LIN {X 0,Y 573.014,Z 552.895,A -85,B 0,C 180,E1 -2253.868,E2 -2253.868} C_VEL
LIN {X 0,Y 572.963,Z 548.948,A -85,B 0,C 180,E1 -2254.926,E2 -2254.926} C_VEL
LIN {X 0,Y 573.068,Z 542.875,A -85,B 0,C 180,E1 -2256.16,E2 -2256.16} C_VEL
LIN {X 0,Y 573.12,Z 536.235,A -85,B 0,C 180,E1 -2257.221,E2 -2257.221} C_VEL
LIN {X 0,Y 573.192,Z 527.989,A -85,B 0,C 180,E1 -2258.284,E2 -2258.284} C_VEL
LIN {X 0,Y 573.32,Z 517.598,A -85,B 0,C 180,E1 -2259.348,E2 -2259.348} C_VEL
LIN {X 0,Y 573.431,Z 507.921,A -85,B 0,C 180,E1 -2260.148,E2 -2260.148} C_VEL
LIN {X 0,Y 573.55,Z 497.399,A -85,B 0,C 180,E1 -2260.855,E2 -2260.855} C_VEL
LIN {X 0,Y 573.653,Z 486.284,A -85,B 0,C 180,E1 -2261.447,E2 -2261.447} C_VEL
LIN {X 0,Y 573.72,Z 473.165,A -85,B 0,C 180,E1 -2261.975,E2 -2261.975} C_VEL
LIN {X 0,Y 573.814,Z 460.51,A -85,B 0,C 180,E1 -2262.332,E2 -2262.332} C_VEL
LIN {X 0,Y 573.909,Z 447.293,A -85,B 0,C 180,E1 -2262.554,E2 -2262.554} C_VEL
LIN {X 0,Y 573.91,Z 350.259,A -85,B 0,C 180,E1 -2263.776,E2 -2263.776} C_VEL
LIN {X 0,Y 573.399,Z 346.611,A -85,B 0,C 180,E1 -2263.851,E2 -2263.851} C_VEL
LIN {X 0,Y 573.569,Z 326.119,A -85,B 0,C 180,E1 -2266.727,E2 -2266.727} C_VEL
LIN {X 0,Y 573.804,Z 305.61,A -85,B 0,C 180,E1 -2269.646,E2 -2269.646} C_VEL
LIN {X 0,Y 574.03,Z 285.748,A -85,B 0,C 180,E1 -2272.495,E2 -2272.495} C_VEL
LIN {X 0,Y 573.588,Z 280.776,A -85,B 0,C 180,E1 -2273.226,E2 -2273.226} C_VEL
LIN {X 0,Y 573.253,Z 279.081,A -85,B 0,C 180,E1 -2273.497,E2 -2273.497} C_VEL
LIN {X 0,Y 573.261,Z 279.08,A -85,B 0,C 180,E1 -2276.19,E2 -2276.19} C_VEL
LIN {X 0,Y 573.237,Z 279.078,A -85,B 0,C 180,E1 -2278.564,E2 -2278.564} C_VEL
LIN {X 0,Y 573.227,Z 279.076,A -85,B 0,C 180,E1 -2280.993,E2 -2280.993} C_VEL
LIN {X 0,Y 573.265,Z 279.071,A -85,B 0,C 180,E1 -2283.524,E2 -2283.524} C_VEL
LIN {X 0,Y 573.216,Z 279.083,A -85,B 0,C 180,E1 -2286.051,E2 -2286.051} C_VEL
LIN {X 0,Y 573.241,Z 279.079,A -85,B 0,C 180,E1 -2288.701,E2 -2288.701} C_VEL
LIN {X 0,Y 573.23,Z 279.075,A -85,B 0,C 180,E1 -2291.593,E2 -2291.593} C_VEL
LIN {X 0,Y 573.222,Z 279.082,A -85,B 0,C 180,E1 -2294.334,E2 -2294.334} C_VEL
LIN {X 0,Y 573.241,Z 279.074,A -85,B 0,C 180,E1 -2297.358,E2 -2297.358} C_VEL
LIN {X 0,Y 573.239,Z 279.077,A -85,B 0,C 180,E1 -2300.392,E2 -2300.392} C_VEL
LIN {X 0,Y 573.252,Z 279.078,A -85,B 0,C 180,E1 -2303.077,E2 -2303.077} C_VEL
LIN {X 0,Y 573.266,Z 279.07,A -85,B 0,C 180,E1 -2305.671,E2 -2305.671} C_VEL
LIN {X 0,Y 573.239,Z 279.074,A -85,B 0,C 180,E1 -2308.184,E2 -2308.184} C_VEL
LIN {X 0,Y 573.263,Z 279.073,A -85,B 0,C 180,E1 -2310.634,E2 -2310.634} C_VEL
LIN {X 0,Y 573.249,Z 279.08,A -85,B 0,C 180,E1 -2313.024,E2 -2313.024} C_VEL
LIN {X 0,Y 573.273,Z 279.077,A -85,B 0,C 180,E1 -2315.366,E2 -2315.366} C_VEL
LIN {X 0,Y 573.227,Z 279.075,A -85,B 0,C 180,E1 -2318.419,E2 -2318.419} C_VEL
LIN {X 0,Y 573.277,Z 279.069,A -85,B 0,C 180,E1 -2320.728,E2 -2320.728} C_VEL
LIN {X 0,Y 573.249,Z 279.08,A -85,B 0,C 180,E1 -2323.622,E2 -2323.622} C_VEL
LIN {X 0,Y 573.271,Z 279.075,A -85,B 0,C 180,E1 -2325.807,E2 -2325.807} C_VEL
LIN {X 0,Y 573.26,Z 279.07,A -85,B 0,C 180,E1 -2328.745,E2 -2328.745} C_VEL
LIN {X 0,Y 573.281,Z 279.074,A -85,B 0,C 180,E1 -2331.54,E2 -2331.54} C_VEL
LIN {X 0,Y 573.288,Z 279.068,A -85,B 0,C 180,E1 -2334.372,E2 -2334.372} C_VEL
LIN {X 0,Y 573.309,Z 279.074,A -85,B 0,C 180,E1 -2337.892,E2 -2337.892} C_VEL
LIN {X 0,Y 573.327,Z 279.063,A -85,B 0,C 180,E1 -2340.702,E2 -2340.702} C_VEL
LIN {X 0,Y 573.236,Z 279.074,A -85,B 0,C 180,E1 -2343.514,E2 -2343.514} C_VEL
LIN {X 0,Y 573.288,Z 279.069,A -85,B 0,C 180,E1 -2345.628,E2 -2345.628} C_VEL
LIN {X 0,Y 573.281,Z 279.075,A -85,B 0,C 180,E1 -2348.459,E2 -2348.459} C_VEL
LIN {X 0,Y 573.269,Z 279.069,A -85,B 0,C 180,E1 -2351.312,E2 -2351.312} C_VEL
LIN {X 0,Y 573.279,Z 279.079,A -85,B 0,C 180,E1 -2354.424,E2 -2354.424} C_VEL
LIN {X 0,Y 573.256,Z 279.073,A -85,B 0,C 180,E1 -2357.112,E2 -2357.112} C_VEL
LIN {X 0,Y 573.25,Z 279.074,A -85,B 0,C 180,E1 -2360.077,E2 -2360.077} C_VEL
LIN {X 0,Y 573.232,Z 279.078,A -85,B 0,C 180,E1 -2363.099,E2 -2363.099} C_VEL
LIN {X 0,Y 573.248,Z 279.076,A -85,B 0,C 180,E1 -2364.382,E2 -2364.382} C_VEL
LIN {X 0,Y 572.62,Z 279.161,A -85,B 0,C 180,E1 -2364.969,E2 -2364.969} C_VEL
LIN {X 0,Y 569.779,Z 279.516,A -85,B 0,C 180,E1 -2365.92,E2 -2365.92} C_VEL
LIN {X 0,Y 567.347,Z 279.815,A -85,B 0,C 180,E1 -2366.686,E2 -2366.686} C_VEL
LIN {X 0,Y 566.292,Z 279.942,A -85,B 0,C 180,E1 -2367.277,E2 -2367.277} C_VEL
LIN {X 0,Y 566.201,Z 279.951,A -85,B 0,C 180,E1 -2367.477,E2 -2367.477} C_VEL
LIN {X 0,Y 566.199,Z 279.95,A -85,B 0,C 180,E1 -2369.769,E2 -2369.769} C_VEL
LIN {X 0,Y 566.201,Z 279.951,A -85,B 0,C 180,E1 -2372.43,E2 -2372.43} C_VEL
LIN {X 0,Y 566.179,Z 279.961,A -85,B 0,C 180,E1 -2374.99,E2 -2374.99} C_VEL
LIN {X 0,Y 566.195,Z 279.957,A -85,B 0,C 180,E1 -2377.461,E2 -2377.461} C_VEL
LIN {X 0,Y 566.206,Z 279.949,A -85,B 0,C 180,E1 -2380.199,E2 -2380.199} C_VEL
LIN {X 0,Y 566.2,Z 279.956,A -85,B 0,C 180,E1 -2383.054,E2 -2383.054} C_VEL
LIN {X 0,Y 566.193,Z 279.953,A -85,B 0,C 180,E1 -2386.049,E2 -2386.049} C_VEL
LIN {X 0,Y 566.203,Z 279.955,A -85,B 0,C 180,E1 -2389.215,E2 -2389.215} C_VEL
LIN {X 0,Y 566.185,Z 279.962,A -85,B 0,C 180,E1 -2391.637,E2 -2391.637} C_VEL
LIN {X 0,Y 566.162,Z 279.957,A -85,B 0,C 180,E1 -2394.308,E2 -2394.308} C_VEL
LIN {X 0,Y 566.205,Z 279.951,A -85,B 0,C 180,E1 -2396.897,E2 -2396.897} C_VEL
LIN {X 0,Y 566.181,Z 279.958,A -85,B 0,C 180,E1 -2399.407,E2 -2399.407} C_VEL
LIN {X 0,Y 566.242,Z 280.056,A -85,B 0,C 180,E1 -2400.897,E2 -2400.897} C_VEL
LIN {X 0,Y 566.45,Z 286.564,A -85,B 0,C 180,E1 -2402.072,E2 -2402.072} C_VEL
LIN {X 0,Y 566.262,Z 302.821,A -85,B 0,C 180,E1 -2405.04,E2 -2405.04} C_VEL
LIN {X 0,Y 566.202,Z 308.373,A -85,B 0,C 180,E1 -2406.045,E2 -2406.045} C_VEL
LIN {X 0,Y 567.204,Z 314.789,A -85,B 0,C 180,E1 -2406.161,E2 -2406.161} C_VEL
LIN {X 0,Y 566.892,Z 414.942,A -85,B 0,C 180,E1 -2407.447,E2 -2407.447} C_VEL
LIN {X 0,Y 566.74,Z 428.708,A -85,B 0,C 180,E1 -2407.776,E2 -2407.776} C_VEL
LIN {X 0,Y 566.676,Z 440.788,A -85,B 0,C 180,E1 -2408.209,E2 -2408.209} C_VEL
LIN {X 0,Y 566.58,Z 452.966,A -85,B 0,C 180,E1 -2408.798,E2 -2408.798} C_VEL
LIN {X 0,Y 566.416,Z 463.929,A -85,B 0,C 180,E1 -2409.481,E2 -2409.481} C_VEL
LIN {X 0,Y 566.302,Z 474.815,A -85,B 0,C 180,E1 -2410.328,E2 -2410.328} C_VEL
LIN {X 0,Y 566.23,Z 483.591,A -85,B 0,C 180,E1 -2411.173,E2 -2411.173} C_VEL
LIN {X 0,Y 566.102,Z 491.649,A -85,B 0,C 180,E1 -2412.105,E2 -2412.105} C_VEL
LIN {X 0,Y 566.039,Z 499.147,A -85,B 0,C 180,E1 -2413.176,E2 -2413.176} C_VEL
LIN {X 0,Y 565.951,Z 504.676,A -85,B 0,C 180,E1 -2414.145,E2 -2414.145} C_VEL
LIN {X 0,Y 565.943,Z 509.72,A -85,B 0,C 180,E1 -2415.252,E2 -2415.252} C_VEL
LIN {X 0,Y 565.898,Z 513.562,A -85,B 0,C 180,E1 -2416.351,E2 -2416.351} C_VEL
LIN {X 0,Y 565.86,Z 515.527,A -85,B 0,C 180,E1 -2417.082,E2 -2417.082} C_VEL
LIN {X 0,Y 565.869,Z 517.042,A -85,B 0,C 180,E1 -2417.811,E2 -2417.811} C_VEL
LIN {X 0,Y 565.901,Z 518.433,A -85,B 0,C 180,E1 -2418.846,E2 -2418.846} C_VEL
LIN {X 0,Y 565.882,Z 518.993,A -85,B 0,C 180,E1 -2419.987,E2 -2419.987} C_VEL
LIN {X 0,Y 565.829,Z 518.818,A -85,B 0,C 180,E1 -2420.708,E2 -2420.708} C_VEL
LIN {X 0,Y 565.851,Z 518.23,A -85,B 0,C 180,E1 -2421.428,E2 -2421.428} C_VEL
LIN {X 0,Y 565.876,Z 517.248,A -85,B 0,C 180,E1 -2422.148,E2 -2422.148} C_VEL
LIN {X 0,Y 565.946,Z 514.44,A -85,B 0,C 180,E1 -2423.44,E2 -2423.44} C_VEL
LIN {X 0,Y 565.921,Z 510.451,A -85,B 0,C 180,E1 -2424.655,E2 -2424.655} C_VEL
LIN {X 0,Y 565.964,Z 505.778,A -85,B 0,C 180,E1 -2425.727,E2 -2425.727} C_VEL
LIN {X 0,Y 566.002,Z 498.771,A -85,B 0,C 180,E1 -2426.975,E2 -2426.975} C_VEL
LIN {X 0,Y 566.065,Z 491.207,A -85,B 0,C 180,E1 -2428.043,E2 -2428.043} C_VEL
LIN {X 0,Y 566.211,Z 481.731,A -85,B 0,C 180,E1 -2429.111,E2 -2429.111} C_VEL
LIN {X 0,Y 566.297,Z 472.006,A -85,B 0,C 180,E1 -2430,E2 -2430} C_VEL
LIN {X 0,Y 566.443,Z 461.142,A -85,B 0,C 180,E1 -2430.799,E2 -2430.799} C_VEL
LIN {X 0,Y 566.641,Z 448.809,A -85,B 0,C 180,E1 -2431.51,E2 -2431.51} C_VEL
LIN {X 0,Y 566.743,Z 436.745,A -85,B 0,C 180,E1 -2432.043,E2 -2432.043} C_VEL
LIN {X 0,Y 566.815,Z 424.109,A -85,B 0,C 180,E1 -2432.442,E2 -2432.442} C_VEL
LIN {X 0,Y 566.945,Z 410.737,A -85,B 0,C 180,E1 -2432.708,E2 -2432.708} C_VEL
LIN {X 0,Y 567.094,Z 313.951,A -85,B 0,C 180,E1 -2433.943,E2 -2433.943} C_VEL
LIN {X 0,Y 566.199,Z 308.359,A -85,B 0,C 180,E1 -2434.048,E2 -2434.048} C_VEL
LIN {X 0,Y 566.374,Z 295.33,A -85,B 0,C 180,E1 -2436.412,E2 -2436.412} C_VEL
LIN {X 0,Y 566.401,Z 281.613,A -85,B 0,C 180,E1 -2438.922,E2 -2438.922} C_VEL
LIN {X 0,Y 566.187,Z 279.958,A -85,B 0,C 180,E1 -2439.241,E2 -2439.241} C_VEL
LIN {X 0,Y 566.192,Z 279.953,A -85,B 0,C 180,E1 -2441.455,E2 -2441.455} C_VEL
LIN {X 0,Y 566.213,Z 279.956,A -85,B 0,C 180,E1 -2444.497,E2 -2444.497} C_VEL
LIN {X 0,Y 566.17,Z 279.954,A -85,B 0,C 180,E1 -2447.332,E2 -2447.332} C_VEL
LIN {X 0,Y 566.2,Z 279.959,A -85,B 0,C 180,E1 -2450.337,E2 -2450.337} C_VEL
LIN {X 0,Y 566.163,Z 279.955,A -85,B 0,C 180,E1 -2453.279,E2 -2453.279} C_VEL
LIN {X 0,Y 566.169,Z 279.954,A -85,B 0,C 180,E1 -2455.75,E2 -2455.75} C_VEL
LIN {X 0,Y 566.149,Z 279.96,A -85,B 0,C 180,E1 -2458.192,E2 -2458.192} C_VEL
LIN {X 0,Y 566.177,Z 279.958,A -85,B 0,C 180,E1 -2461.074,E2 -2461.074} C_VEL
LIN {X 0,Y 566.192,Z 279.951,A -85,B 0,C 180,E1 -2463.731,E2 -2463.731} C_VEL
LIN {X 0,Y 566.193,Z 279.956,A -85,B 0,C 180,E1 -2466.569,E2 -2466.569} C_VEL
LIN {X 0,Y 566.204,Z 279.95,A -85,B 0,C 180,E1 -2469.684,E2 -2469.684} C_VEL
LIN {X 0,Y 566.166,Z 279.954,A -85,B 0,C 180,E1 -2472.09,E2 -2472.09} C_VEL
LIN {X 0,Y 566.161,Z 279.964,A -85,B 0,C 180,E1 -2475.036,E2 -2475.036} C_VEL
LIN {X 0,Y 566.18,Z 279.953,A -85,B 0,C 180,E1 -2477.91,E2 -2477.91} C_VEL
LIN {X 0,Y 566.203,Z 279.952,A -85,B 0,C 180,E1 -2480.725,E2 -2480.725} C_VEL
LIN {X 0,Y 566.175,Z 279.957,A -85,B 0,C 180,E1 -2483.788,E2 -2483.788} C_VEL
LIN {X 0,Y 566.203,Z 279.95,A -85,B 0,C 180,E1 -2486.265,E2 -2486.265} C_VEL
LIN {X 0,Y 566.18,Z 279.955,A -85,B 0,C 180,E1 -2488.923,E2 -2488.923} C_VEL
LIN {X 0,Y 566.178,Z 279.958,A -85,B 0,C 180,E1 -2491.856,E2 -2491.856} C_VEL
LIN {X 0,Y 566.203,Z 279.951,A -85,B 0,C 180,E1 -2494.251,E2 -2494.251} C_VEL
LIN {X 0,Y 566.16,Z 279.955,A -85,B 0,C 180,E1 -2496.719,E2 -2496.719} C_VEL
LIN {X 0,Y 566.198,Z 279.959,A -85,B 0,C 180,E1 -2499.662,E2 -2499.662} C_VEL
LIN {X 0,Y 566.192,Z 279.951,A -85,B 0,C 180,E1 -2502.668,E2 -2502.668} C_VEL
LIN {X 0,Y 566.211,Z 279.954,A -85,B 0,C 180,E1 -2505.626,E2 -2505.626} C_VEL
LIN {X 0,Y 566.225,Z 279.948,A -85,B 0,C 180,E1 -2508.675,E2 -2508.675} C_VEL
LIN {X 0,Y 566.218,Z 279.949,A -85,B 0,C 180,E1 -2511.434,E2 -2511.434} C_VEL
LIN {X 0,Y 566.253,Z 279.952,A -85,B 0,C 180,E1 -2514.302,E2 -2514.302} C_VEL
LIN {X 0,Y 566.268,Z 279.946,A -85,B 0,C 180,E1 -2517.866,E2 -2517.866} C_VEL
LIN {X 0,Y 566.299,Z 279.942,A -85,B 0,C 180,E1 -2520.711,E2 -2520.711} C_VEL
LIN {X 0,Y 566.269,Z 279.945,A -85,B 0,C 180,E1 -2522.846,E2 -2522.846} C_VEL
LIN {X 0,Y 566.249,Z 279.944,A -85,B 0,C 180,E1 -2525.699,E2 -2525.699} C_VEL
LIN {X 0,Y 566.239,Z 279.956,A -85,B 0,C 180,E1 -2528.566,E2 -2528.566} C_VEL
LIN {X 0,Y 566.243,Z 279.945,A -85,B 0,C 180,E1 -2531.454,E2 -2531.454} C_VEL
LIN {X 0,Y 566.225,Z 279.954,A -85,B 0,C 180,E1 -2534.507,E2 -2534.507} C_VEL
LIN {X 0,Y 566.191,Z 279.953,A -85,B 0,C 180,E1 -2537.332,E2 -2537.332} C_VEL
LIN {X 0,Y 566.205,Z 279.952,A -85,B 0,C 180,E1 -2540.338,E2 -2540.338} C_VEL
LIN {X 0,Y 566.182,Z 279.955,A -85,B 0,C 180,E1 -2543.404,E2 -2543.404} C_VEL
LIN {X 0,Y 566.218,Z 279.948,A -85,B 0,C 180,E1 -2545.749,E2 -2545.749} C_VEL
LIN {X 0,Y 566.195,Z 279.951,A -85,B 0,C 180,E1 -2548.203,E2 -2548.203} C_VEL
LIN {X 0,Y 566.187,Z 279.954,A -85,B 0,C 180,E1 -2550.593,E2 -2550.593} C_VEL
LIN {X 0,Y 566.223,Z 279.956,A -85,B 0,C 180,E1 -2553.102,E2 -2553.102} C_VEL
LIN {X 0,Y 566.2,Z 279.95,A -85,B 0,C 180,E1 -2556.216,E2 -2556.216} C_VEL
LIN {X 0,Y 566.216,Z 279.957,A -85,B 0,C 180,E1 -2559.274,E2 -2559.274} C_VEL
LIN {X 0,Y 566.209,Z 279.95,A -85,B 0,C 180,E1 -2562.088,E2 -2562.088} C_VEL
LIN {X 0,Y 566.169,Z 279.957,A -85,B 0,C 180,E1 -2565.037,E2 -2565.037} C_VEL
LIN {X 0,Y 566.215,Z 279.951,A -85,B 0,C 180,E1 -2568.137,E2 -2568.137} C_VEL
LIN {X 0,Y 566.211,Z 279.949,A -85,B 0,C 180,E1 -2570.727,E2 -2570.727} C_VEL
LIN {X 0,Y 566.182,Z 279.963,A -85,B 0,C 180,E1 -2573.789,E2 -2573.789} C_VEL
LIN {X 0,Y 566.21,Z 279.952,A -85,B 0,C 180,E1 -2576.267,E2 -2576.267} C_VEL
LIN {X 0,Y 566.189,Z 279.951,A -85,B 0,C 180,E1 -2578.924,E2 -2578.924} C_VEL
LIN {X 0,Y 566.229,Z 279.957,A -85,B 0,C 180,E1 -2581.859,E2 -2581.859} C_VEL
LIN {X 0,Y 566.237,Z 279.948,A -85,B 0,C 180,E1 -2585.04,E2 -2585.04} C_VEL
LIN {X 0,Y 566.24,Z 280.067,A -85,B 0,C 180,E1 -2586.381,E2 -2586.381} C_VEL
LIN {X 0,Y 567.09,Z 285.538,A -85,B 0,C 180,E1 -2587.215,E2 -2587.215} C_VEL
LIN {X 0,Y 566.868,Z 306.731,A -85,B 0,C 180,E1 -2590.274,E2 -2590.274} C_VEL
LIN {X 0,Y 566.599,Z 327.553,A -85,B 0,C 180,E1 -2593.267,E2 -2593.267} C_VEL
LIN {X 0,Y 566.389,Z 346.617,A -85,B 0,C 180,E1 -2595.975,E2 -2595.975} C_VEL
LIN {X 0,Y 567.201,Z 352.33,A -85,B 0,C 180,E1 -2596.084,E2 -2596.084} C_VEL
LIN {X 0,Y 566.953,Z 454.975,A -85,B 0,C 180,E1 -2597.403,E2 -2597.403} C_VEL
LIN {X 0,Y 566.837,Z 468.237,A -85,B 0,C 180,E1 -2597.719,E2 -2597.719} C_VEL
LIN {X 0,Y 566.722,Z 480.39,A -85,B 0,C 180,E1 -2598.148,E2 -2598.148} C_VEL
LIN {X 0,Y 566.626,Z 492.163,A -85,B 0,C 180,E1 -2598.709,E2 -2598.709} C_VEL
LIN {X 0,Y 566.458,Z 504.206,A -85,B 0,C 180,E1 -2599.456,E2 -2599.456} C_VEL
LIN {X 0,Y 566.32,Z 514.609,A -85,B 0,C 180,E1 -2600.266,E2 -2600.266} C_VEL
LIN {X 0,Y 566.205,Z 523.088,A -85,B 0,C 180,E1 -2601.075,E2 -2601.075} C_VEL
LIN {X 0,Y 566.111,Z 530.965,A -85,B 0,C 180,E1 -2601.972,E2 -2601.972} C_VEL
LIN {X 0,Y 566.003,Z 538.625,A -85,B 0,C 180,E1 -2603.047,E2 -2603.047} C_VEL
LIN {X 0,Y 566.004,Z 545.682,A -85,B 0,C 180,E1 -2604.3,E2 -2604.3} C_VEL
LIN {X 0,Y 565.933,Z 550.374,A -85,B 0,C 180,E1 -2605.371,E2 -2605.371} C_VEL
LIN {X 0,Y 565.926,Z 553.959,A -85,B 0,C 180,E1 -2606.44,E2 -2606.44} C_VEL
LIN {X 0,Y 565.878,Z 555.809,A -85,B 0,C 180,E1 -2607.153,E2 -2607.153} C_VEL
LIN {X 0,Y 565.845,Z 558.185,A -85,B 0,C 180,E1 -2608.577,E2 -2608.577} C_VEL
LIN {X 0,Y 565.839,Z 559,A -85,B 0,C 180,E1 -2610,E2 -2610} C_VEL
LIN {X 0,Y 565.845,Z 558.185,A -85,B 0,C 180,E1 -2611.424,E2 -2611.424} C_VEL
LIN {X 0,Y 565.878,Z 555.809,A -85,B 0,C 180,E1 -2612.848,E2 -2612.848} C_VEL
LIN {X 0,Y 565.926,Z 552.895,A -85,B 0,C 180,E1 -2613.917,E2 -2613.917} C_VEL
LIN {X 0,Y 565.878,Z 548.947,A -85,B 0,C 180,E1 -2614.988,E2 -2614.988} C_VEL
LIN {X 0,Y 565.994,Z 542.875,A -85,B 0,C 180,E1 -2616.238,E2 -2616.238} C_VEL
LIN {X 0,Y 566.052,Z 536.235,A -85,B 0,C 180,E1 -2617.312,E2 -2617.312} C_VEL
LIN {X 0,Y 566.141,Z 527.989,A -85,B 0,C 180,E1 -2618.388,E2 -2618.388} C_VEL
LIN {X 0,Y 566.254,Z 519.536,A -85,B 0,C 180,E1 -2619.285,E2 -2619.285} C_VEL
LIN {X 0,Y 566.416,Z 509.093,A -85,B 0,C 180,E1 -2620.184,E2 -2620.184} C_VEL
LIN {X 0,Y 566.571,Z 497.699,A -85,B 0,C 180,E1 -2620.971,E2 -2620.971} C_VEL
LIN {X 0,Y 566.693,Z 485.881,A -85,B 0,C 180,E1 -2621.608,E2 -2621.608} C_VEL
LIN {X 0,Y 566.79,Z 473.163,A -85,B 0,C 180,E1 -2622.124,E2 -2622.124} C_VEL
LIN {X 0,Y 566.877,Z 460.509,A -85,B 0,C 180,E1 -2622.485,E2 -2622.485} C_VEL
LIN {X 0,Y 566.977,Z 447.293,A -85,B 0,C 180,E1 -2622.71,E2 -2622.71} C_VEL
LIN {X 0,Y 567.066,Z 351.263,A -85,B 0,C 180,E1 -2623.933,E2 -2623.933} C_VEL
LIN {X 0,Y 566.407,Z 346.611,A -85,B 0,C 180,E1 -2624.025,E2 -2624.025} C_VEL
LIN {X 0,Y 566.607,Z 324.039,A -85,B 0,C 180,E1 -2627.238,E2 -2627.238} C_VEL
LIN {X 0,Y 566.869,Z 303.946,A -85,B 0,C 180,E1 -2630.123,E2 -2630.123} C_VEL
LIN {X 0,Y 567.055,Z 285.451,A -85,B 0,C 180,E1 -2632.787,E2 -2632.787} C_VEL
LIN {X 0,Y 566.215,Z 279.958,A -85,B 0,C 180,E1 -2633.645,E2 -2633.645} C_VEL
LIN {X 0,Y 566.21,Z 279.958,A -85,B 0,C 180,E1 -2635.749,E2 -2635.749} C_VEL
LIN {X 0,Y 566.206,Z 279.96,A -85,B 0,C 180,E1 -2638.202,E2 -2638.202} C_VEL
LIN {X 0,Y 566.193,Z 279.953,A -85,B 0,C 180,E1 -2641.076,E2 -2641.076} C_VEL
LIN {X 0,Y 566.213,Z 279.951,A -85,B 0,C 180,E1 -2643.734,E2 -2643.734} C_VEL
LIN {X 0,Y 566.201,Z 279.957,A -85,B 0,C 180,E1 -2646.57,E2 -2646.57} C_VEL
LIN {X 0,Y 566.215,Z 279.949,A -85,B 0,C 180,E1 -2649.685,E2 -2649.685} C_VEL
LIN {X 0,Y 566.202,Z 279.955,A -85,B 0,C 180,E1 -2652.917,E2 -2652.917} C_VEL
LIN {X 0,Y 566.194,Z 279.953,A -85,B 0,C 180,E1 -2656.049,E2 -2656.049} C_VEL
LIN {X 0,Y 566.204,Z 279.952,A -85,B 0,C 180,E1 -2659.214,E2 -2659.214} C_VEL
LIN {X 0,Y 566.186,Z 279.952,A -85,B 0,C 180,E1 -2661.637,E2 -2661.637} C_VEL
LIN {X 0,Y 566.162,Z 279.957,A -85,B 0,C 180,E1 -2664.308,E2 -2664.308} C_VEL
LIN {X 0,Y 566.219,Z 279.957,A -85,B 0,C 180,E1 -2666.898,E2 -2666.898} C_VEL
LIN {X 0,Y 566.18,Z 279.957,A -85,B 0,C 180,E1 -2669.407,E2 -2669.407} C_VEL
LIN {X 0,Y 566.21,Z 279.95,A -85,B 0,C 180,E1 -2671.857,E2 -2671.857} C_VEL
LIN {X 0,Y 566.212,Z 279.948,A -85,B 0,C 180,E1 -2674.251,E2 -2674.251} C_VEL
LIN {X 0,Y 566.172,Z 279.956,A -85,B 0,C 180,E1 -2676.718,E2 -2676.718} C_VEL
LIN {X 0,Y 566.212,Z 279.954,A -85,B 0,C 180,E1 -2679.663,E2 -2679.663} C_VEL
LIN {X 0,Y 566.198,Z 279.95,A -85,B 0,C 180,E1 -2682.668,E2 -2682.668} C_VEL
LIN {X 0,Y 566.232,Z 279.955,A -85,B 0,C 180,E1 -2685.627,E2 -2685.627} C_VEL
LIN {X 0,Y 566.232,Z 279.945,A -85,B 0,C 180,E1 -2688.675,E2 -2688.675} C_VEL
LIN {X 0,Y 566.225,Z 279.951,A -85,B 0,C 180,E1 -2691.434,E2 -2691.434} C_VEL
LIN {X 0,Y 566.256,Z 279.945,A -85,B 0,C 180,E1 -2694.302,E2 -2694.302} C_VEL
LIN {X 0,Y 566.28,Z 279.949,A -85,B 0,C 180,E1 -2697.866,E2 -2697.866} C_VEL
LIN {X 0,Y 566.298,Z 279.938,A -85,B 0,C 180,E1 -2700.711,E2 -2700.711} C_VEL
LIN {X 0,Y 566.269,Z 279.941,A -85,B 0,C 180,E1 -2702.845,E2 -2702.845} C_VEL
LIN {X 0,Y 566.256,Z 279.945,A -85,B 0,C 180,E1 -2705.698,E2 -2705.698} C_VEL
LIN {X 0,Y 566.225,Z 279.952,A -85,B 0,C 180,E1 -2708.566,E2 -2708.566} C_VEL
LIN {X 0,Y 566.24,Z 279.945,A -85,B 0,C 180,E1 -2711.454,E2 -2711.454} C_VEL
LIN {X 0,Y 566.232,Z 279.956,A -85,B 0,C 180,E1 -2714.507,E2 -2714.507} C_VEL
LIN {X 0,Y 566.197,Z 279.951,A -85,B 0,C 180,E1 -2717.332,E2 -2717.332} C_VEL
LIN {X 0,Y 566.211,Z 279.954,A -85,B 0,C 180,E1 -2720.337,E2 -2720.337} C_VEL
LIN {X 0,Y 566.187,Z 279.953,A -85,B 0,C 180,E1 -2723.404,E2 -2723.404} C_VEL
LIN {X 0,Y 566.212,Z 279.948,A -85,B 0,C 180,E1 -2725.749,E2 -2725.749} C_VEL
LIN {X 0,Y 566.201,Z 279.951,A -85,B 0,C 180,E1 -2727.477,E2 -2727.477} C_VEL
LIN {X 0,Y 565.521,Z 280.036,A -85,B 0,C 180,E1 -2728.071,E2 -2728.071} C_VEL
LIN {X 0,Y 562.655,Z 280.4,A -85,B 0,C 180,E1 -2729.034,E2 -2729.034} C_VEL
LIN {X 0,Y 560.246,Z 280.696,A -85,B 0,C 180,E1 -2729.81,E2 -2729.81} C_VEL
LIN {X 0,Y 559.218,Z 280.822,A -85,B 0,C 180,E1 -2730.409,E2 -2730.409} C_VEL
LIN {X 0,Y 559.138,Z 280.833,A -85,B 0,C 180,E1 -2730.611,E2 -2730.611} C_VEL
LIN {X 0,Y 559.161,Z 280.829,A -85,B 0,C 180,E1 -2733.575,E2 -2733.575} C_VEL
LIN {X 0,Y 559.145,Z 280.83,A -85,B 0,C 180,E1 -2736.445,E2 -2736.445} C_VEL
LIN {X 0,Y 559.173,Z 280.831,A -85,B 0,C 180,E1 -2738.934,E2 -2738.934} C_VEL
LIN {X 0,Y 559.166,Z 280.83,A -85,B 0,C 180,E1 -2741.77,E2 -2741.77} C_VEL
LIN {X 0,Y 559.131,Z 280.832,A -85,B 0,C 180,E1 -2744.74,E2 -2744.74} C_VEL
LIN {X 0,Y 559.157,Z 280.834,A -85,B 0,C 180,E1 -2747.256,E2 -2747.256} C_VEL
LIN {X 0,Y 559.179,Z 280.828,A -85,B 0,C 180,E1 -2750.135,E2 -2750.135} C_VEL
LIN {X 0,Y 559.14,Z 280.831,A -85,B 0,C 180,E1 -2752.892,E2 -2752.892} C_VEL
LIN {X 0,Y 559.165,Z 280.834,A -85,B 0,C 180,E1 -2756.051,E2 -2756.051} C_VEL
LIN {X 0,Y 559.156,Z 280.83,A -85,B 0,C 180,E1 -2758.981,E2 -2758.981} C_VEL
LIN {X 0,Y 559.19,Z 280.895,A -85,B 0,C 180,E1 -2760.881,E2 -2760.881} C_VEL
LIN {X 0,Y 559.409,Z 286.774,A -85,B 0,C 180,E1 -2761.935,E2 -2761.935} C_VEL
LIN {X 0,Y 559.282,Z 302.509,A -85,B 0,C 180,E1 -2764.791,E2 -2764.791} C_VEL
LIN {X 0,Y 559.202,Z 308.562,A -85,B 0,C 180,E1 -2765.877,E2 -2765.877} C_VEL
LIN {X 0,Y 560.314,Z 315.979,A -85,B 0,C 180,E1 -2766.002,E2 -2766.002} C_VEL
LIN {X 0,Y 559.961,Z 415.434,A -85,B 0,C 180,E1 -2767.298,E2 -2767.298} C_VEL
LIN {X 0,Y 559.796,Z 429.032,A -85,B 0,C 180,E1 -2767.632,E2 -2767.632} C_VEL
LIN {X 0,Y 559.735,Z 441.208,A -85,B 0,C 180,E1 -2768.077,E2 -2768.077} C_VEL
LIN {X 0,Y 559.613,Z 452.707,A -85,B 0,C 180,E1 -2768.641,E2 -2768.641} C_VEL
LIN {X 0,Y 559.422,Z 463.384,A -85,B 0,C 180,E1 -2769.309,E2 -2769.309} C_VEL
LIN {X 0,Y 559.311,Z 474.377,A -85,B 0,C 180,E1 -2770.168,E2 -2770.168} C_VEL
LIN {X 0,Y 559.173,Z 484.133,A -85,B 0,C 180,E1 -2771.117,E2 -2771.117} C_VEL
LIN {X 0,Y 559.039,Z 492.071,A -85,B 0,C 180,E1 -2772.061,E2 -2772.061} C_VEL
LIN {X 0,Y 558.957,Z 499.773,A -85,B 0,C 180,E1 -2773.19,E2 -2773.19} C_VEL
LIN {X 0,Y 558.865,Z 505.89,A -85,B 0,C 180,E1 -2774.313,E2 -2774.313} C_VEL
LIN {X 0,Y 558.826,Z 511.113,A -85,B 0,C 180,E1 -2775.553,E2 -2775.553} C_VEL
LIN {X 0,Y 558.763,Z 515.209,A -85,B 0,C 180,E1 -2776.915,E2 -2776.915} C_VEL
LIN {X 0,Y 558.777,Z 516.805,A -85,B 0,C 180,E1 -2777.654,E2 -2777.654} C_VEL
LIN {X 0,Y 558.799,Z 518.416,A -85,B 0,C 180,E1 -2778.815,E2 -2778.815} C_VEL
LIN {X 0,Y 558.778,Z 518.966,A -85,B 0,C 180,E1 -2779.858,E2 -2779.858} C_VEL
LIN {X 0,Y 558.74,Z 518.885,A -85,B 0,C 180,E1 -2780.589,E2 -2780.589} C_VEL
LIN {X 0,Y 558.765,Z 518.368,A -85,B 0,C 180,E1 -2781.319,E2 -2781.319} C_VEL
LIN {X 0,Y 558.795,Z 517.445,A -85,B 0,C 180,E1 -2782.047,E2 -2782.047} C_VEL
LIN {X 0,Y 558.844,Z 514.489,A -85,B 0,C 180,E1 -2783.464,E2 -2783.464} C_VEL
LIN {X 0,Y 558.845,Z 510.936,A -85,B 0,C 180,E1 -2784.588,E2 -2784.588} C_VEL
LIN {X 0,Y 558.892,Z 506.399,A -85,B 0,C 180,E1 -2785.673,E2 -2785.673} C_VEL
LIN {X 0,Y 558.906,Z 499.551,A -85,B 0,C 180,E1 -2786.936,E2 -2786.936} C_VEL
LIN {X 0,Y 559,Z 492.156,A -85,B 0,C 180,E1 -2788.018,E2 -2788.018} C_VEL
LIN {X 0,Y 559.146,Z 484.633,A -85,B 0,C 180,E1 -2788.919,E2 -2788.919} C_VEL
LIN {X 0,Y 559.24,Z 475.571,A -85,B 0,C 180,E1 -2789.82,E2 -2789.82} C_VEL
LIN {X 0,Y 559.355,Z 465.543,A -85,B 0,C 180,E1 -2790.63,E2 -2790.63} C_VEL
LIN {X 0,Y 559.61,Z 454.423,A -85,B 0,C 180,E1 -2791.349,E2 -2791.349} C_VEL
LIN {X 0,Y 559.751,Z 443.962,A -85,B 0,C 180,E1 -2791.888,E2 -2791.888} C_VEL
LIN {X 0,Y 559.843,Z 431.433,A -85,B 0,C 180,E1 -2792.383,E2 -2792.383} C_VEL
LIN {X 0,Y 559.98,Z 419.001,A -85,B 0,C 180,E1 -2792.72,E2 -2792.72} C_VEL
LIN {X 0,Y 560.068,Z 403.28,A -85,B 0,C 180,E1 -2792.967,E2 -2792.967} C_VEL
LIN {X 0,Y 560.118,Z 314.336,A -85,B 0,C 180,E1 -2794.114,E2 -2794.114} C_VEL
LIN {X 0,Y 559.172,Z 308.323,A -85,B 0,C 180,E1 -2794.234,E2 -2794.234} C_VEL
LIN {X 0,Y 559.351,Z 294.875,A -85,B 0,C 180,E1 -2796.702,E2 -2796.702} C_VEL
LIN {X 0,Y 559.39,Z 283.104,A -85,B 0,C 180,E1 -2798.853,E2 -2798.853} C_VEL
LIN {X 0,Y 559.141,Z 280.836,A -85,B 0,C 180,E1 -2799.313,E2 -2799.313} C_VEL
LIN {X 0,Y 559.155,Z 280.831,A -85,B 0,C 180,E1 -2801.601,E2 -2801.601} C_VEL
LIN {X 0,Y 559.16,Z 280.833,A -85,B 0,C 180,E1 -2804.579,E2 -2804.579} C_VEL
LIN {X 0,Y 559.12,Z 280.832,A -85,B 0,C 180,E1 -2807.558,E2 -2807.558} C_VEL
LIN {X 0,Y 559.171,Z 280.834,A -85,B 0,C 180,E1 -2810.604,E2 -2810.604} C_VEL
LIN {X 0,Y 559.116,Z 280.833,A -85,B 0,C 180,E1 -2813.717,E2 -2813.717} C_VEL
LIN {X 0,Y 559.14,Z 280.832,A -85,B 0,C 180,E1 -2816.098,E2 -2816.098} C_VEL
LIN {X 0,Y 559.107,Z 280.842,A -85,B 0,C 180,E1 -2818.532,E2 -2818.532} C_VEL
LIN {X 0,Y 559.133,Z 280.833,A -85,B 0,C 180,E1 -2821.271,E2 -2821.271} C_VEL
LIN {X 0,Y 559.149,Z 280.829,A -85,B 0,C 180,E1 -2823.946,E2 -2823.946} C_VEL
LIN {X 0,Y 559.135,Z 280.837,A -85,B 0,C 180,E1 -2827.108,E2 -2827.108} C_VEL
LIN {X 0,Y 559.152,Z 280.828,A -85,B 0,C 180,E1 -2829.94,E2 -2829.94} C_VEL
LIN {X 0,Y 559.141,Z 280.835,A -85,B 0,C 180,E1 -2832.744,E2 -2832.744} C_VEL
LIN {X 0,Y 559.122,Z 280.84,A -85,B 0,C 180,E1 -2835.259,E2 -2835.259} C_VEL
LIN {X 0,Y 559.153,Z 280.828,A -85,B 0,C 180,E1 -2838.229,E2 -2838.229} C_VEL
LIN {X 0,Y 559.165,Z 280.836,A -85,B 0,C 180,E1 -2841.191,E2 -2841.191} C_VEL
LIN {X 0,Y 559.13,Z 280.834,A -85,B 0,C 180,E1 -2843.789,E2 -2843.789} C_VEL
LIN {X 0,Y 559.15,Z 280.828,A -85,B 0,C 180,E1 -2846.424,E2 -2846.424} C_VEL
LIN {X 0,Y 559.145,Z 280.832,A -85,B 0,C 180,E1 -2848.98,E2 -2848.98} C_VEL
LIN {X 0,Y 559.159,Z 280.837,A -85,B 0,C 180,E1 -2851.618,E2 -2851.618} C_VEL
LIN {X 0,Y 559.167,Z 280.826,A -85,B 0,C 180,E1 -2854.701,E2 -2854.701} C_VEL
LIN {X 0,Y 559.131,Z 280.839,A -85,B 0,C 180,E1 -2857.847,E2 -2857.847} C_VEL
LIN {X 0,Y 559.183,Z 280.825,A -85,B 0,C 180,E1 -2860.494,E2 -2860.494} C_VEL
LIN {X 0,Y 559.171,Z 280.827,A -85,B 0,C 180,E1 -2863.197,E2 -2863.197} C_VEL
LIN {X 0,Y 559.154,Z 280.834,A -85,B 0,C 180,E1 -2866.184,E2 -2866.184} C_VEL
LIN {X 0,Y 559.196,Z 280.824,A -85,B 0,C 180,E1 -2868.604,E2 -2868.604} C_VEL
LIN {X 0,Y 559.177,Z 280.826,A -85,B 0,C 180,E1 -2871.326,E2 -2871.326} C_VEL
LIN {X 0,Y 559.219,Z 280.829,A -85,B 0,C 180,E1 -2874.23,E2 -2874.23} C_VEL
LIN {X 0,Y 559.24,Z 280.821,A -85,B 0,C 180,E1 -2877.839,E2 -2877.839} C_VEL
LIN {X 0,Y 559.268,Z 280.818,A -85,B 0,C 180,E1 -2880.72,E2 -2880.72} C_VEL
LIN {X 0,Y 559.235,Z 280.821,A -85,B 0,C 180,E1 -2882.881,E2 -2882.881} C_VEL
LIN {X 0,Y 559.218,Z 280.821,A -85,B 0,C 180,E1 -2885.77,E2 -2885.77} C_VEL
LIN {X 0,Y 559.194,Z 280.831,A -85,B 0,C 180,E1 -2888.674,E2 -2888.674} C_VEL
LIN {X 0,Y 559.201,Z 280.822,A -85,B 0,C 180,E1 -2891.601,E2 -2891.601} C_VEL
LIN {X 0,Y 559.191,Z 280.832,A -85,B 0,C 180,E1 -2894.596,E2 -2894.596} C_VEL
LIN {X 0,Y 559.151,Z 280.829,A -85,B 0,C 180,E1 -2897.557,E2 -2897.557} C_VEL
LIN {X 0,Y 559.164,Z 280.827,A -85,B 0,C 180,E1 -2899.838,E2 -2899.838} C_VEL
LIN {X 0,Y 559.133,Z 280.831,A -85,B 0,C 180,E1 -2902.153,E2 -2902.153} C_VEL
LIN {X 0,Y 559.172,Z 280.833,A -85,B 0,C 180,E1 -2905.188,E2 -2905.188} C_VEL
LIN {X 0,Y 559.177,Z 280.826,A -85,B 0,C 180,E1 -2907.713,E2 -2907.713} C_VEL
LIN {X 0,Y 559.162,Z 280.827,A -85,B 0,C 180,E1 -2910.182,E2 -2910.182} C_VEL
LIN {X 0,Y 559.169,Z 280.829,A -85,B 0,C 180,E1 -2912.715,E2 -2912.715} C_VEL
LIN {X 0,Y 559.139,Z 280.839,A -85,B 0,C 180,E1 -2915.323,E2 -2915.323} C_VEL
LIN {X 0,Y 559.129,Z 280.832,A -85,B 0,C 180,E1 -2918.018,E2 -2918.018} C_VEL
LIN {X 0,Y 559.172,Z 280.827,A -85,B 0,C 180,E1 -2920.811,E2 -2920.811} C_VEL
LIN {X 0,Y 559.155,Z 280.834,A -85,B 0,C 180,E1 -2923.733,E2 -2923.733} C_VEL
LIN {X 0,Y 559.143,Z 280.83,A -85,B 0,C 180,E1 -2926.804,E2 -2926.804} C_VEL
LIN {X 0,Y 559.156,Z 280.831,A -85,B 0,C 180,E1 -2929.189,E2 -2929.189} C_VEL
LIN {X 0,Y 559.13,Z 280.836,A -85,B 0,C 180,E1 -2931.983,E2 -2931.983} C_VEL
LIN {X 0,Y 559.129,Z 280.831,A -85,B 0,C 180,E1 -2934.788,E2 -2934.788} C_VEL
LIN {X 0,Y 559.154,Z 280.831,A -85,B 0,C 180,E1 -2937.365,E2 -2937.365} C_VEL
LIN {X 0,Y 559.148,Z 280.837,A -85,B 0,C 180,E1 -2940.143,E2 -2940.143} C_VEL
LIN {X 0,Y 559.169,Z 280.827,A -85,B 0,C 180,E1 -2943.098,E2 -2943.098} C_VEL
LIN {X 0,Y 559.182,Z 280.836,A -85,B 0,C 180,E1 -2946.089,E2 -2946.089} C_VEL
LIN {X 0,Y 559.197,Z 280.971,A -85,B 0,C 180,E1 -2946.237,E2 -2946.237} C_VEL
LIN {X 0,Y 560.144,Z 286.611,A -85,B 0,C 180,E1 -2947.112,E2 -2947.112} C_VEL
LIN {X 0,Y 559.899,Z 306.356,A -85,B 0,C 180,E1 -2949.999,E2 -2949.999} C_VEL
LIN {X 0,Y 559.622,Z 326.688,A -85,B 0,C 180,E1 -2952.927,E2 -2952.927} C_VEL
LIN {X 0,Y 559.395,Z 346.617,A -85,B 0,C 180,E1 -2955.796,E2 -2955.796} C_VEL
LIN {X 0,Y 560.278,Z 354.343,A -85,B 0,C 180,E1 -2955.935,E2 -2955.935} C_VEL
LIN {X 0,Y 560.036,Z 454.975,A -85,B 0,C 180,E1 -2957.245,E2 -2957.245} C_VEL
LIN {X 0,Y 559.914,Z 468.236,A -85,B 0,C 180,E1 -2957.565,E2 -2957.565} C_VEL
LIN {X 0,Y 559.764,Z 480.392,A -85,B 0,C 180,E1 -2957.999,E2 -2957.999} C_VEL
LIN {X 0,Y 559.668,Z 491.822,A -85,B 0,C 180,E1 -2958.548,E2 -2958.548} C_VEL
LIN {X 0,Y 559.491,Z 502.912,A -85,B 0,C 180,E1 -2959.231,E2 -2959.231} C_VEL
LIN {X 0,Y 559.308,Z 513.544,A -85,B 0,C 180,E1 -2960.051,E2 -2960.051} C_VEL
LIN {X 0,Y 559.161,Z 523.101,A -85,B 0,C 180,E1 -2960.961,E2 -2960.961} C_VEL
LIN {X 0,Y 559.046,Z 530.965,A -85,B 0,C 180,E1 -2961.87,E2 -2961.87} C_VEL
LIN {X 0,Y 558.943,Z 538.625,A -85,B 0,C 180,E1 -2962.959,E2 -2962.959} C_VEL
LIN {X 0,Y 558.936,Z 545.682,A -85,B 0,C 180,E1 -2964.227,E2 -2964.227} C_VEL
LIN {X 0,Y 558.826,Z 550.374,A -85,B 0,C 180,E1 -2965.312,E2 -2965.312} C_VEL
LIN {X 0,Y 558.836,Z 553.959,A -85,B 0,C 180,E1 -2966.395,E2 -2966.395} C_VEL
LIN {X 0,Y 558.799,Z 555.808,A -85,B 0,C 180,E1 -2967.117,E2 -2967.117} C_VEL
LIN {X 0,Y 558.745,Z 558.184,A -85,B 0,C 180,E1 -2968.559,E2 -2968.559} C_VEL
LIN {X 0,Y 558.74,Z 559,A -85,B 0,C 180,E1 -2970,E2 -2970} C_VEL
LIN {X 0,Y 558.745,Z 558.185,A -85,B 0,C 180,E1 -2971.442,E2 -2971.442} C_VEL
LIN {X 0,Y 558.799,Z 555.809,A -85,B 0,C 180,E1 -2972.884,E2 -2972.884} C_VEL
LIN {X 0,Y 558.844,Z 552.894,A -85,B 0,C 180,E1 -2973.967,E2 -2973.967} C_VEL
LIN {X 0,Y 558.798,Z 548.947,A -85,B 0,C 180,E1 -2975.051,E2 -2975.051} C_VEL
LIN {X 0,Y 558.925,Z 543.866,A -85,B 0,C 180,E1 -2976.136,E2 -2976.136} C_VEL
LIN {X 0,Y 558.978,Z 537.465,A -85,B 0,C 180,E1 -2977.223,E2 -2977.223} C_VEL
LIN {X 0,Y 559.091,Z 529.475,A -85,B 0,C 180,E1 -2978.312,E2 -2978.312} C_VEL
LIN {X 0,Y 559.185,Z 521.332,A -85,B 0,C 180,E1 -2979.221,E2 -2979.221} C_VEL
LIN {X 0,Y 559.347,Z 511.396,A -85,B 0,C 180,E1 -2980.132,E2 -2980.132} C_VEL
LIN {X 0,Y 559.57,Z 500.375,A -85,B 0,C 180,E1 -2980.938,E2 -2980.938} C_VEL
LIN {X 0,Y 559.672,Z 488.455,A -85,B 0,C 180,E1 -2981.628,E2 -2981.628} C_VEL
LIN {X 0,Y 559.795,Z 475.761,A -85,B 0,C 180,E1 -2982.185,E2 -2982.185} C_VEL
LIN {X 0,Y 559.927,Z 462.337,A -85,B 0,C 180,E1 -2982.597,E2 -2982.597} C_VEL
LIN {X 0,Y 560.098,Z 449.069,A -85,B 0,C 180,E1 -2982.846,E2 -2982.846} C_VEL
LIN {X 0,Y 560.224,Z 352.269,A -85,B 0,C 180,E1 -2984.093,E2 -2984.093} C_VEL
LIN {X 0,Y 559.41,Z 346.611,A -85,B 0,C 180,E1 -2984.204,E2 -2984.204} C_VEL
LIN {X 0,Y 559.62,Z 324.689,A -85,B 0,C 180,E1 -2987.359,E2 -2987.359} C_VEL
LIN {X 0,Y 559.892,Z 304.973,A -85,B 0,C 180,E1 -2990.194,E2 -2990.194} C_VEL
LIN {X 0,Y 560.099,Z 286.482,A -85,B 0,C 180,E1 -2992.891,E2 -2992.891} C_VEL
LIN {X 0,Y 559.178,Z 280.836,A -85,B 0,C 180,E1 -2993.764,E2 -2993.764} C_VEL
LIN {X 0,Y 559.177,Z 280.836,A -85,B 0,C 180,E1 -2996.097,E2 -2996.097} C_VEL
LIN {X 0,Y 559.165,Z 280.832,A -85,B 0,C 180,E1 -2998.53,E2 -2998.53} C_VEL
LIN {X 0,Y 559.148,Z 280.831,A -85,B 0,C 180,E1 -3001.273,E2 -3001.273} C_VEL
LIN {X 0,Y 559.166,Z 280.832,A -85,B 0,C 180,E1 -3003.949,E2 -3003.949} C_VEL
LIN {X 0,Y 559.142,Z 280.831,A -85,B 0,C 180,E1 -3007.108,E2 -3007.108} C_VEL
LIN {X 0,Y 559.161,Z 280.83,A -85,B 0,C 180,E1 -3009.941,E2 -3009.941} C_VEL
LIN {X 0,Y 559.158,Z 280.835,A -85,B 0,C 180,E1 -3012.744,E2 -3012.744} C_VEL
LIN {X 0,Y 559.148,Z 280.829,A -85,B 0,C 180,E1 -3015.761,E2 -3015.761} C_VEL
LIN {X 0,Y 559.163,Z 280.83,A -85,B 0,C 180,E1 -3018.23,E2 -3018.23} C_VEL
LIN {X 0,Y 559.174,Z 280.829,A -85,B 0,C 180,E1 -3021.191,E2 -3021.191} C_VEL
LIN {X 0,Y 559.138,Z 280.83,A -85,B 0,C 180,E1 -3023.789,E2 -3023.789} C_VEL
LIN {X 0,Y 559.162,Z 280.828,A -85,B 0,C 180,E1 -3026.425,E2 -3026.425} C_VEL
LIN {X 0,Y 559.155,Z 280.838,A -85,B 0,C 180,E1 -3028.98,E2 -3028.98} C_VEL
LIN {X 0,Y 559.167,Z 280.829,A -85,B 0,C 180,E1 -3031.619,E2 -3031.619} C_VEL
LIN {X 0,Y 559.18,Z 280.825,A -85,B 0,C 180,E1 -3033.903,E2 -3033.903} C_VEL
LIN {X 0,Y 559.141,Z 280.83,A -85,B 0,C 180,E1 -3036.571,E2 -3036.571} C_VEL
LIN {X 0,Y 559.178,Z 280.835,A -85,B 0,C 180,E1 -3039.395,E2 -3039.395} C_VEL
LIN {X 0,Y 559.145,Z 280.835,A -85,B 0,C 180,E1 -3041.686,E2 -3041.686} C_VEL
LIN {X 0,Y 559.164,Z 280.829,A -85,B 0,C 180,E1 -3043.948,E2 -3043.948} C_VEL
LIN {X 0,Y 559.17,Z 280.827,A -85,B 0,C 180,E1 -3046.184,E2 -3046.184} C_VEL
LIN {X 0,Y 559.191,Z 280.825,A -85,B 0,C 180,E1 -3049.133,E2 -3049.133} C_VEL
LIN {X 0,Y 559.201,Z 280.827,A -85,B 0,C 180,E1 -3052.053,E2 -3052.053} C_VEL
LIN {X 0,Y 559.249,Z 280.814,A -85,B 0,C 180,E1 -3054.953,E2 -3054.953} C_VEL
LIN {X 0,Y 559.251,Z 280.824,A -85,B 0,C 180,E1 -3057.839,E2 -3057.839} C_VEL
LIN {X 0,Y 559.268,Z 280.814,A -85,B 0,C 180,E1 -3060.72,E2 -3060.72} C_VEL
LIN {X 0,Y 559.236,Z 280.816,A -85,B 0,C 180,E1 -3062.881,E2 -3062.881} C_VEL
LIN {X 0,Y 559.225,Z 280.822,A -85,B 0,C 180,E1 -3065.77,E2 -3065.77} C_VEL
LIN {X 0,Y 559.184,Z 280.828,A -85,B 0,C 180,E1 -3068.674,E2 -3068.674} C_VEL
LIN {X 0,Y 559.203,Z 280.822,A -85,B 0,C 180,E1 -3071.6,E2 -3071.6} C_VEL
LIN {X 0,Y 559.198,Z 280.831,A -85,B 0,C 180,E1 -3074.596,E2 -3074.596} C_VEL
LIN {X 0,Y 559.157,Z 280.827,A -85,B 0,C 180,E1 -3077.557,E2 -3077.557} C_VEL
LIN {X 0,Y 559.17,Z 280.826,A -85,B 0,C 180,E1 -3079.837,E2 -3079.837} C_VEL
LIN {X 0,Y 559.139,Z 280.832,A -85,B 0,C 180,E1 -3082.153,E2 -3082.153} C_VEL
LIN {X 0,Y 559.177,Z 280.829,A -85,B 0,C 180,E1 -3085.187,E2 -3085.187} C_VEL
LIN {X 0,Y 559.155,Z 280.827,A -85,B 0,C 180,E1 -3087.714,E2 -3087.714} C_VEL
LIN {X 0,Y 559.138,Z 280.833,A -85,B 0,C 180,E1 -3090.611,E2 -3090.611} C_VEL
LIN {X 0,Y 558.476,Z 280.921,A -85,B 0,C 180,E1 -3091.213,E2 -3091.213} C_VEL
LIN {X 0,Y 555.614,Z 281.278,A -85,B 0,C 180,E1 -3092.189,E2 -3092.189} C_VEL
LIN {X 0,Y 553.201,Z 281.578,A -85,B 0,C 180,E1 -3092.974,E2 -3092.974} C_VEL
LIN {X 0,Y 552.182,Z 281.699,A -85,B 0,C 180,E1 -3093.581,E2 -3093.581} C_VEL
LIN {X 0,Y 552.108,Z 281.706,A -85,B 0,C 180,E1 -3093.786,E2 -3093.786} C_VEL
LIN {X 0,Y 552.104,Z 281.71,A -85,B 0,C 180,E1 -3096.747,E2 -3096.747} C_VEL
LIN {X 0,Y 552.128,Z 281.708,A -85,B 0,C 180,E1 -3099.527,E2 -3099.527} C_VEL
LIN {X 0,Y 552.129,Z 281.703,A -85,B 0,C 180,E1 -3102.426,E2 -3102.426} C_VEL
LIN {X 0,Y 552.091,Z 281.717,A -85,B 0,C 180,E1 -3105.562,E2 -3105.562} C_VEL
LIN {X 0,Y 552.121,Z 281.704,A -85,B 0,C 180,E1 -3108.554,E2 -3108.554} C_VEL
LIN {X 0,Y 552.117,Z 281.712,A -85,B 0,C 180,E1 -3111.411,E2 -3111.411} C_VEL
LIN {X 0,Y 552.085,Z 281.712,A -85,B 0,C 180,E1 -3114.156,E2 -3114.156} C_VEL
LIN {X 0,Y 552.112,Z 281.707,A -85,B 0,C 180,E1 -3116.814,E2 -3116.814} C_VEL
LIN {X 0,Y 552.103,Z 281.712,A -85,B 0,C 180,E1 -3119.391,E2 -3119.391} C_VEL
LIN {X 0,Y 552.173,Z 281.902,A -85,B 0,C 180,E1 -3120.867,E2 -3120.867} C_VEL
LIN {X 0,Y 552.378,Z 289.017,A -85,B 0,C 180,E1 -3122.123,E2 -3122.123} C_VEL
LIN {X 0,Y 552.253,Z 304.213,A -85,B 0,C 180,E1 -3124.894,E2 -3124.894} C_VEL
LIN {X 0,Y 552.175,Z 308.442,A -85,B 0,C 180,E1 -3125.684,E2 -3125.684} C_VEL
LIN {X 0,Y 553.442,Z 317.036,A -85,B 0,C 180,E1 -3125.837,E2 -3125.837} C_VEL
LIN {X 0,Y 553.041,Z 414.718,A -85,B 0,C 180,E1 -3127.121,E2 -3127.121} C_VEL
LIN {X 0,Y 552.934,Z 427.797,A -85,B 0,C 180,E1 -3127.437,E2 -3127.437} C_VEL
LIN {X 0,Y 552.766,Z 440.097,A -85,B 0,C 180,E1 -3127.878,E2 -3127.878} C_VEL
LIN {X 0,Y 552.646,Z 452.032,A -85,B 0,C 180,E1 -3128.457,E2 -3128.457} C_VEL
LIN {X 0,Y 552.441,Z 462.842,A -85,B 0,C 180,E1 -3129.132,E2 -3129.132} C_VEL
LIN {X 0,Y 552.29,Z 472.805,A -85,B 0,C 180,E1 -3129.905,E2 -3129.905} C_VEL
LIN {X 0,Y 552.118,Z 482.888,A -85,B 0,C 180,E1 -3130.866,E2 -3130.866} C_VEL
LIN {X 0,Y 551.98,Z 491.069,A -85,B 0,C 180,E1 -3131.824,E2 -3131.824} C_VEL
LIN {X 0,Y 551.908,Z 498.964,A -85,B 0,C 180,E1 -3132.969,E2 -3132.969} C_VEL
LIN {X 0,Y 551.793,Z 505.236,A -85,B 0,C 180,E1 -3134.107,E2 -3134.107} C_VEL
LIN {X 0,Y 551.772,Z 510.16,A -85,B 0,C 180,E1 -3135.241,E2 -3135.241} C_VEL
LIN {X 0,Y 551.715,Z 513.891,A -85,B 0,C 180,E1 -3136.369,E2 -3136.369} C_VEL
LIN {X 0,Y 551.667,Z 516.547,A -85,B 0,C 180,E1 -3137.492,E2 -3137.492} C_VEL
LIN {X 0,Y 551.71,Z 518.391,A -85,B 0,C 180,E1 -3138.775,E2 -3138.775} C_VEL
LIN {X 0,Y 551.675,Z 518.937,A -85,B 0,C 180,E1 -3139.726,E2 -3139.726} C_VEL
LIN {X 0,Y 551.669,Z 518.498,A -85,B 0,C 180,E1 -3141.206,E2 -3141.206} C_VEL
LIN {X 0,Y 551.694,Z 517.642,A -85,B 0,C 180,E1 -3141.944,E2 -3141.944} C_VEL
LIN {X 0,Y 551.744,Z 514.713,A -85,B 0,C 180,E1 -3143.417,E2 -3143.417} C_VEL
LIN {X 0,Y 551.769,Z 511.372,A -85,B 0,C 180,E1 -3144.518,E2 -3144.518} C_VEL
LIN {X 0,Y 551.799,Z 506.968,A -85,B 0,C 180,E1 -3145.617,E2 -3145.617} C_VEL
LIN {X 0,Y 551.813,Z 501.39,A -85,B 0,C 180,E1 -3146.714,E2 -3146.714} C_VEL
LIN {X 0,Y 551.91,Z 494.44,A -85,B 0,C 180,E1 -3147.81,E2 -3147.81} C_VEL
LIN {X 0,Y 552.085,Z 485.763,A -85,B 0,C 180,E1 -3148.906,E2 -3148.906} C_VEL
LIN {X 0,Y 552.213,Z 476.923,A -85,B 0,C 180,E1 -3149.817,E2 -3149.817} C_VEL
LIN {X 0,Y 552.356,Z 466.048,A -85,B 0,C 180,E1 -3150.729,E2 -3150.729} C_VEL
LIN {X 0,Y 552.626,Z 455.045,A -85,B 0,C 180,E1 -3151.457,E2 -3151.457} C_VEL
LIN {X 0,Y 552.796,Z 442.792,A -85,B 0,C 180,E1 -3152.094,E2 -3152.094} C_VEL
LIN {X 0,Y 552.912,Z 431.161,A -85,B 0,C 180,E1 -3152.549,E2 -3152.549} C_VEL
LIN {X 0,Y 553.059,Z 418.54,A -85,B 0,C 180,E1 -3152.89,E2 -3152.89} C_VEL
LIN {X 0,Y 553.168,Z 400.792,A -85,B 0,C 180,E1 -3153.163,E2 -3153.163} C_VEL
LIN {X 0,Y 553.287,Z 315.35,A -85,B 0,C 180,E1 -3154.279,E2 -3154.279} C_VEL
LIN {X 0,Y 552.143,Z 308.346,A -85,B 0,C 180,E1 -3154.425,E2 -3154.425} C_VEL
LIN {X 0,Y 552.303,Z 294.387,A -85,B 0,C 180,E1 -3157.001,E2 -3157.001} C_VEL
LIN {X 0,Y 552.36,Z 283.711,A -85,B 0,C 180,E1 -3158.966,E2 -3158.966} C_VEL
LIN {X 0,Y 552.096,Z 281.714,A -85,B 0,C 180,E1 -3159.386,E2 -3159.386} C_VEL
LIN {X 0,Y 552.101,Z 281.711,A -85,B 0,C 180,E1 -3161.751,E2 -3161.751} C_VEL
LIN {X 0,Y 552.122,Z 281.707,A -85,B 0,C 180,E1 -3164.748,E2 -3164.748} C_VEL
LIN {X 0,Y 552.08,Z 281.711,A -85,B 0,C 180,E1 -3167.789,E2 -3167.789} C_VEL
LIN {X 0,Y 552.118,Z 281.709,A -85,B 0,C 180,E1 -3170.101,E2 -3170.101} C_VEL
LIN {X 0,Y 552.085,Z 281.718,A -85,B 0,C 180,E1 -3172.45,E2 -3172.45} C_VEL
LIN {X 0,Y 552.075,Z 281.71,A -85,B 0,C 180,E1 -3175.332,E2 -3175.332} C_VEL
LIN {X 0,Y 552.056,Z 281.714,A -85,B 0,C 180,E1 -3178.1,E2 -3178.1} C_VEL
LIN {X 0,Y 552.084,Z 281.717,A -85,B 0,C 180,E1 -3180.609,E2 -3180.609} C_VEL
LIN {X 0,Y 552.099,Z 281.711,A -85,B 0,C 180,E1 -3183.186,E2 -3183.186} C_VEL
LIN {X 0,Y 552.08,Z 281.709,A -85,B 0,C 180,E1 -3185.843,E2 -3185.843} C_VEL
LIN {X 0,Y 552.108,Z 281.71,A -85,B 0,C 180,E1 -3188.589,E2 -3188.589} C_VEL
LIN {X 0,Y 552.07,Z 281.714,A -85,B 0,C 180,E1 -3191.449,E2 -3191.449} C_VEL
LIN {X 0,Y 552.086,Z 281.709,A -85,B 0,C 180,E1 -3194.437,E2 -3194.437} C_VEL
LIN {X 0,Y 552.102,Z 281.71,A -85,B 0,C 180,E1 -3197.586,E2 -3197.586} C_VEL
LIN {X 0,Y 552.12,Z 281.705,A -85,B 0,C 180,E1 -3200.472,E2 -3200.472} C_VEL
LIN {X 0,Y 552.098,Z 281.717,A -85,B 0,C 180,E1 -3203.316,E2 -3203.316} C_VEL
LIN {X 0,Y 552.117,Z 281.707,A -85,B 0,C 180,E1 -3205.938,E2 -3205.938} C_VEL
LIN {X 0,Y 552.111,Z 281.705,A -85,B 0,C 180,E1 -3208.54,E2 -3208.54} C_VEL
LIN {X 0,Y 552.114,Z 281.713,A -85,B 0,C 180,E1 -3211.438,E2 -3211.438} C_VEL
LIN {X 0,Y 552.119,Z 281.705,A -85,B 0,C 180,E1 -3214.355,E2 -3214.355} C_VEL
LIN {X 0,Y 552.087,Z 281.708,A -85,B 0,C 180,E1 -3216.757,E2 -3216.757} C_VEL
LIN {X 0,Y 552.109,Z 281.707,A -85,B 0,C 180,E1 -3219.119,E2 -3219.119} C_VEL
LIN {X 0,Y 552.114,Z 281.709,A -85,B 0,C 180,E1 -3221.444,E2 -3221.444} C_VEL
LIN {X 0,Y 552.105,Z 281.714,A -85,B 0,C 180,E1 -3223.737,E2 -3223.737} C_VEL
LIN {X 0,Y 552.12,Z 281.714,A -85,B 0,C 180,E1 -3226.004,E2 -3226.004} C_VEL
LIN {X 0,Y 552.152,Z 281.7,A -85,B 0,C 180,E1 -3228.993,E2 -3228.993} C_VEL
LIN {X 0,Y 552.15,Z 281.708,A -85,B 0,C 180,E1 -3231.951,E2 -3231.951} C_VEL
LIN {X 0,Y 552.217,Z 281.693,A -85,B 0,C 180,E1 -3234.889,E2 -3234.889} C_VEL
LIN {X 0,Y 552.211,Z 281.696,A -85,B 0,C 180,E1 -3237.812,E2 -3237.812} C_VEL
LIN {X 0,Y 552.237,Z 281.693,A -85,B 0,C 180,E1 -3240.729,E2 -3240.729} C_VEL
LIN {X 0,Y 552.201,Z 281.696,A -85,B 0,C 180,E1 -3242.918,E2 -3242.918} C_VEL
LIN {X 0,Y 552.188,Z 281.697,A -85,B 0,C 180,E1 -3245.844,E2 -3245.844} C_VEL
LIN {X 0,Y 552.162,Z 281.705,A -85,B 0,C 180,E1 -3248.786,E2 -3248.786} C_VEL
LIN {X 0,Y 552.156,Z 281.7,A -85,B 0,C 180,E1 -3251.751,E2 -3251.751} C_VEL
LIN {X 0,Y 552.128,Z 281.713,A -85,B 0,C 180,E1 -3254.749,E2 -3254.749} C_VEL
LIN {X 0,Y 552.102,Z 281.706,A -85,B 0,C 180,E1 -3257.789,E2 -3257.789} C_VEL
LIN {X 0,Y 552.123,Z 281.704,A -85,B 0,C 180,E1 -3260.102,E2 -3260.102} C_VEL
LIN {X 0,Y 552.088,Z 281.711,A -85,B 0,C 180,E1 -3262.451,E2 -3262.451} C_VEL
LIN {X 0,Y 552.15,Z 281.705,A -85,B 0,C 180,E1 -3265.351,E2 -3265.351} C_VEL
LIN {X 0,Y 552.114,Z 281.705,A -85,B 0,C 180,E1 -3268.098,E2 -3268.098} C_VEL
LIN {X 0,Y 552.108,Z 281.708,A -85,B 0,C 180,E1 -3270.609,E2 -3270.609} C_VEL
LIN {X 0,Y 552.117,Z 281.715,A -85,B 0,C 180,E1 -3273.186,E2 -3273.186} C_VEL
LIN {X 0,Y 552.097,Z 281.709,A -85,B 0,C 180,E1 -3275.843,E2 -3275.843} C_VEL
LIN {X 0,Y 552.12,Z 281.71,A -85,B 0,C 180,E1 -3279.063,E2 -3279.063} C_VEL
LIN {X 0,Y 552.135,Z 281.713,A -85,B 0,C 180,E1 -3281.445,E2 -3281.445} C_VEL
LIN {X 0,Y 552.091,Z 281.708,A -85,B 0,C 180,E1 -3284.533,E2 -3284.533} C_VEL
LIN {X 0,Y 552.127,Z 281.714,A -85,B 0,C 180,E1 -3287.585,E2 -3287.585} C_VEL
LIN {X 0,Y 552.126,Z 281.704,A -85,B 0,C 180,E1 -3290.474,E2 -3290.474} C_VEL
LIN {X 0,Y 552.104,Z 281.71,A -85,B 0,C 180,E1 -3293.318,E2 -3293.318} C_VEL
LIN {X 0,Y 552.125,Z 281.712,A -85,B 0,C 180,E1 -3295.94,E2 -3295.94} C_VEL
LIN {X 0,Y 552.118,Z 281.706,A -85,B 0,C 180,E1 -3298.541,E2 -3298.541} C_VEL
LIN {X 0,Y 552.124,Z 281.708,A -85,B 0,C 180,E1 -3301.439,E2 -3301.439} C_VEL
LIN {X 0,Y 552.13,Z 281.712,A -85,B 0,C 180,E1 -3304.357,E2 -3304.357} C_VEL
LIN {X 0,Y 552.17,Z 281.832,A -85,B 0,C 180,E1 -3306.085,E2 -3306.085} C_VEL
LIN {X 0,Y 553.226,Z 288.992,A -85,B 0,C 180,E1 -3307.204,E2 -3307.204} C_VEL
LIN {X 0,Y 552.893,Z 308.997,A -85,B 0,C 180,E1 -3310.159,E2 -3310.159} C_VEL
LIN {X 0,Y 552.614,Z 328.438,A -85,B 0,C 180,E1 -3312.992,E2 -3312.992} C_VEL
LIN {X 0,Y 552.372,Z 346.711,A -85,B 0,C 180,E1 -3315.626,E2 -3315.626} C_VEL
LIN {X 0,Y 553.414,Z 354.829,A -85,B 0,C 180,E1 -3315.763,E2 -3315.763} C_VEL
LIN {X 0,Y 553.111,Z 454.974,A -85,B 0,C 180,E1 -3317.083,E2 -3317.083} C_VEL
LIN {X 0,Y 552.994,Z 468.236,A -85,B 0,C 180,E1 -3317.407,E2 -3317.407} C_VEL
LIN {X 0,Y 552.839,Z 480.383,A -85,B 0,C 180,E1 -3317.846,E2 -3317.846} C_VEL
LIN {X 0,Y 552.689,Z 492.669,A -85,B 0,C 180,E1 -3318.45,E2 -3318.45} C_VEL
LIN {X 0,Y 552.487,Z 504.202,A -85,B 0,C 180,E1 -3319.186,E2 -3319.186} C_VEL
LIN {X 0,Y 552.294,Z 514.612,A -85,B 0,C 180,E1 -3320.016,E2 -3320.016} C_VEL
LIN {X 0,Y 552.125,Z 523.114,A -85,B 0,C 180,E1 -3320.845,E2 -3320.845} C_VEL
LIN {X 0,Y 552.008,Z 530.965,A -85,B 0,C 180,E1 -3321.766,E2 -3321.766} C_VEL
LIN {X 0,Y 551.889,Z 538.625,A -85,B 0,C 180,E1 -3322.868,E2 -3322.868} C_VEL
LIN {X 0,Y 551.868,Z 545.682,A -85,B 0,C 180,E1 -3324.153,E2 -3324.153} C_VEL
LIN {X 0,Y 551.725,Z 550.375,A -85,B 0,C 180,E1 -3325.251,E2 -3325.251} C_VEL
LIN {X 0,Y 551.75,Z 553.959,A -85,B 0,C 180,E1 -3326.349,E2 -3326.349} C_VEL
LIN {X 0,Y 551.723,Z 555.808,A -85,B 0,C 180,E1 -3327.08,E2 -3327.08} C_VEL
LIN {X 0,Y 551.645,Z 558.183,A -85,B 0,C 180,E1 -3328.54,E2 -3328.54} C_VEL
LIN {X 0,Y 551.64,Z 559,A -85,B 0,C 180,E1 -3330,E2 -3330} C_VEL
LIN {X 0,Y 551.645,Z 558.184,A -85,B 0,C 180,E1 -3331.46,E2 -3331.46} C_VEL
LIN {X 0,Y 551.723,Z 555.809,A -85,B 0,C 180,E1 -3332.921,E2 -3332.921} C_VEL
LIN {X 0,Y 551.764,Z 552.894,A -85,B 0,C 180,E1 -3334.017,E2 -3334.017} C_VEL
LIN {X 0,Y 551.724,Z 548.947,A -85,B 0,C 180,E1 -3335.116,E2 -3335.116} C_VEL
LIN {X 0,Y 551.827,Z 543.178,A -85,B 0,C 180,E1 -3336.343,E2 -3336.343} C_VEL
LIN {X 0,Y 551.927,Z 536.234,A -85,B 0,C 180,E1 -3337.5,E2 -3337.5} C_VEL
LIN {X 0,Y 552.064,Z 527.99,A -85,B 0,C 180,E1 -3338.603,E2 -3338.603} C_VEL
LIN {X 0,Y 552.223,Z 519.537,A -85,B 0,C 180,E1 -3339.523,E2 -3339.523} C_VEL
LIN {X 0,Y 552.406,Z 509.089,A -85,B 0,C 180,E1 -3340.445,E2 -3340.445} C_VEL
LIN {X 0,Y 552.61,Z 498.186,A -85,B 0,C 180,E1 -3341.22,E2 -3341.22} C_VEL
LIN {X 0,Y 552.752,Z 487.4,A -85,B 0,C 180,E1 -3341.831,E2 -3341.831} C_VEL
LIN {X 0,Y 552.865,Z 475.758,A -85,B 0,C 180,E1 -3342.341,E2 -3342.341} C_VEL
LIN {X 0,Y 553.006,Z 462.336,A -85,B 0,C 180,E1 -3342.757,E2 -3342.757} C_VEL
LIN {X 0,Y 553.183,Z 449.069,A -85,B 0,C 180,E1 -3343.01,E2 -3343.01} C_VEL
LIN {X 0,Y 553.257,Z 352.314,A -85,B 0,C 180,E1 -3344.274,E2 -3344.274} C_VEL
LIN {X 0,Y 552.383,Z 346.655,A -85,B 0,C 180,E1 -3344.382,E2 -3344.382} C_VEL
LIN {X 0,Y 552.602,Z 326.786,A -85,B 0,C 180,E1 -3347.241,E2 -3347.241} C_VEL
LIN {X 0,Y 552.921,Z 306.006,A -85,B 0,C 180,E1 -3350.265,E2 -3350.265} C_VEL
LIN {X 0,Y 553.15,Z 287.513,A -85,B 0,C 180,E1 -3352.998,E2 -3352.998} C_VEL
LIN {X 0,Y 552.151,Z 281.711,A -85,B 0,C 180,E1 -3353.916,E2 -3353.916} C_VEL
LIN {X 0,Y 552.136,Z 281.705,A -85,B 0,C 180,E1 -3356.999,E2 -3356.999} C_VEL
LIN {X 0,Y 552.119,Z 281.716,A -85,B 0,C 180,E1 -3360.05,E2 -3360.05} C_VEL
LIN {X 0,Y 552.113,Z 281.707,A -85,B 0,C 180,E1 -3362.846,E2 -3362.846} C_VEL
LIN {X 0,Y 552.077,Z 281.711,A -85,B 0,C 180,E1 -3365.439,E2 -3365.439} C_VEL
LIN {X 0,Y 552.097,Z 281.711,A -85,B 0,C 180,E1 -3367.885,E2 -3367.885} C_VEL
LIN {X 0,Y 552.109,Z 281.716,A -85,B 0,C 180,E1 -3370.481,E2 -3370.481} C_VEL
LIN {X 0,Y 552.107,Z 281.707,A -85,B 0,C 180,E1 -3373.423,E2 -3373.423} C_VEL
LIN {X 0,Y 552.107,Z 281.716,A -85,B 0,C 180,E1 -3376.576,E2 -3376.576} C_VEL
LIN {X 0,Y 552.108,Z 281.706,A -85,B 0,C 180,E1 -3379.519,E2 -3379.519} C_VEL
LIN {X 0,Y 552.092,Z 281.711,A -85,B 0,C 180,E1 -3382.336,E2 -3382.336} C_VEL
LIN {X 0,Y 552.083,Z 281.716,A -85,B 0,C 180,E1 -3385.051,E2 -3385.051} C_VEL
LIN {X 0,Y 552.114,Z 281.706,A -85,B 0,C 180,E1 -3387.681,E2 -3387.681} C_VEL
LIN {X 0,Y 552.111,Z 281.705,A -85,B 0,C 180,E1 -3390.235,E2 -3390.235} C_VEL
LIN {X 0,Y 552.137,Z 281.71,A -85,B 0,C 180,E1 -3393,E2 -3393} C_VEL
LIN {X 0,Y 552.113,Z 281.714,A -85,B 0,C 180,E1 -3395.161,E2 -3395.161} C_VEL
LIN {X 0,Y 552.124,Z 281.703,A -85,B 0,C 180,E1 -3398.337,E2 -3398.337} C_VEL
LIN {X 0,Y 552.155,Z 281.7,A -85,B 0,C 180,E1 -3400.674,E2 -3400.674} C_VEL
LIN {X 0,Y 552.115,Z 281.711,A -85,B 0,C 180,E1 -3403.737,E2 -3403.737} C_VEL
LIN {X 0,Y 552.133,Z 281.705,A -85,B 0,C 180,E1 -3406.004,E2 -3406.004} C_VEL
LIN {X 0,Y 552.159,Z 281.7,A -85,B 0,C 180,E1 -3408.993,E2 -3408.993} C_VEL
LIN {X 0,Y 552.155,Z 281.706,A -85,B 0,C 180,E1 -3411.951,E2 -3411.951} C_VEL
LIN {X 0,Y 552.224,Z 281.689,A -85,B 0,C 180,E1 -3414.889,E2 -3414.889} C_VEL
LIN {X 0,Y 552.222,Z 281.699,A -85,B 0,C 180,E1 -3417.812,E2 -3417.812} C_VEL
LIN {X 0,Y 552.239,Z 281.69,A -85,B 0,C 180,E1 -3420.729,E2 -3420.729} C_VEL
LIN {X 0,Y 552.202,Z 281.692,A -85,B 0,C 180,E1 -3422.918,E2 -3422.918} C_VEL
LIN {X 0,Y 552.195,Z 281.699,A -85,B 0,C 180,E1 -3425.844,E2 -3425.844} C_VEL
LIN {X 0,Y 552.155,Z 281.702,A -85,B 0,C 180,E1 -3428.786,E2 -3428.786} C_VEL
LIN {X 0,Y 552.16,Z 281.7,A -85,B 0,C 180,E1 -3431.75,E2 -3431.75} C_VEL
LIN {X 0,Y 552.134,Z 281.708,A -85,B 0,C 180,E1 -3434.748,E2 -3434.748} C_VEL
LIN {X 0,Y 552.108,Z 281.706,A -85,B 0,C 180,E1 -3437.789,E2 -3437.789} C_VEL
LIN {X 0,Y 552.129,Z 281.705,A -85,B 0,C 180,E1 -3440.101,E2 -3440.101} C_VEL
LIN {X 0,Y 552.094,Z 281.713,A -85,B 0,C 180,E1 -3442.451,E2 -3442.451} C_VEL
LIN {X 0,Y 552.154,Z 281.702,A -85,B 0,C 180,E1 -3445.351,E2 -3445.351} C_VEL
LIN {X 0,Y 552.108,Z 281.705,A -85,B 0,C 180,E1 -3448.098,E2 -3448.098} C_VEL
LIN {X 0,Y 552.101,Z 281.711,A -85,B 0,C 180,E1 -3450.609,E2 -3450.609} C_VEL
LIN {X 0,Y 552.113,Z 281.713,A -85,B 0,C 180,E1 -3453.186,E2 -3453.186} C_VEL
LIN {X 0,Y 552.108,Z 281.706,A -85,B 0,C 180,E1 -3453.786,E2 -3453.786} C_VEL
LIN {X 0,Y 551.473,Z 281.786,A -85,B 0,C 180,E1 -3454.395,E2 -3454.395} C_VEL
LIN {X 0,Y 548.651,Z 282.142,A -85,B 0,C 180,E1 -3455.383,E2 -3455.383} C_VEL
LIN {X 0,Y 546.23,Z 282.444,A -85,B 0,C 180,E1 -3456.178,E2 -3456.178} C_VEL
LIN {X 0,Y 545.162,Z 282.577,A -85,B 0,C 180,E1 -3456.792,E2 -3456.792} C_VEL
LIN {X 0,Y 545.061,Z 282.59,A -85,B 0,C 180,E1 -3457,E2 -3457} C_VEL
LIN {X 0,Y 545.065,Z 282.583,A -85,B 0,C 180,E1 -3460.143,E2 -3460.143} C_VEL
LIN {X 0,Y 545.077,Z 282.588,A -85,B 0,C 180,E1 -3463.107,E2 -3463.107} C_VEL
LIN {X 0,Y 545.048,Z 282.586,A -85,B 0,C 180,E1 -3466.226,E2 -3466.226} C_VEL
LIN {X 0,Y 545.081,Z 282.583,A -85,B 0,C 180,E1 -3468.886,E2 -3468.886} C_VEL
LIN {X 0,Y 545.052,Z 282.592,A -85,B 0,C 180,E1 -3471.763,E2 -3471.763} C_VEL
LIN {X 0,Y 545.036,Z 282.588,A -85,B 0,C 180,E1 -3474.532,E2 -3474.532} C_VEL
LIN {X 0,Y 545.066,Z 282.587,A -85,B 0,C 180,E1 -3477.211,E2 -3477.211} C_VEL
LIN {X 0,Y 545.064,Z 282.595,A -85,B 0,C 180,E1 -3479.811,E2 -3479.811} C_VEL
LIN {X 0,Y 545.127,Z 282.628,A -85,B 0,C 180,E1 -3480.777,E2 -3480.777} C_VEL
LIN {X 0,Y 545.351,Z 289.128,A -85,B 0,C 180,E1 -3481.941,E2 -3481.941} C_VEL
LIN {X 0,Y 545.218,Z 300.471,A -85,B 0,C 180,E1 -3484.007,E2 -3484.007} C_VEL
LIN {X 0,Y 545.177,Z 308.493,A -85,B 0,C 180,E1 -3485.485,E2 -3485.485} C_VEL
LIN {X 0,Y 546.577,Z 317.145,A -85,B 0,C 180,E1 -3485.653,E2 -3485.653} C_VEL
LIN {X 0,Y 546.13,Z 415.45,A -85,B 0,C 180,E1 -3486.965,E2 -3486.965} C_VEL
LIN {X 0,Y 545.979,Z 429.125,A -85,B 0,C 180,E1 -3487.309,E2 -3487.309} C_VEL
LIN {X 0,Y 545.863,Z 441.845,A -85,B 0,C 180,E1 -3487.788,E2 -3487.788} C_VEL
LIN {X 0,Y 545.679,Z 453.193,A -85,B 0,C 180,E1 -3488.366,E2 -3488.366} C_VEL
LIN {X 0,Y 545.456,Z 463.77,A -85,B 0,C 180,E1 -3489.05,E2 -3489.05} C_VEL
LIN {X 0,Y 545.282,Z 473.29,A -85,B 0,C 180,E1 -3489.809,E2 -3489.809} C_VEL
LIN {X 0,Y 545.093,Z 483.467,A -85,B 0,C 180,E1 -3490.805,E2 -3490.805} C_VEL
LIN {X 0,Y 544.913,Z 492.911,A -85,B 0,C 180,E1 -3491.968,E2 -3491.968} C_VEL
LIN {X 0,Y 544.789,Z 500.462,A -85,B 0,C 180,E1 -3493.126,E2 -3493.126} C_VEL
LIN {X 0,Y 544.7,Z 506.437,A -85,B 0,C 180,E1 -3494.279,E2 -3494.279} C_VEL
LIN {X 0,Y 544.678,Z 511.005,A -85,B 0,C 180,E1 -3495.404,E2 -3495.404} C_VEL
LIN {X 0,Y 544.627,Z 514.57,A -85,B 0,C 180,E1 -3496.569,E2 -3496.569} C_VEL
LIN {X 0,Y 544.581,Z 516.287,A -85,B 0,C 180,E1 -3497.327,E2 -3497.327} C_VEL
LIN {X 0,Y 544.621,Z 518.366,A -85,B 0,C 180,E1 -3498.735,E2 -3498.735} C_VEL
LIN {X 0,Y 544.579,Z 518.908,A -85,B 0,C 180,E1 -3499.591,E2 -3499.591} C_VEL
LIN {X 0,Y 544.581,Z 518.942,A -85,B 0,C 180,E1 -3500.342,E2 -3500.342} C_VEL
LIN {X 0,Y 544.61,Z 517.832,A -85,B 0,C 180,E1 -3501.839,E2 -3501.839} C_VEL
LIN {X 0,Y 544.603,Z 516.633,A -85,B 0,C 180,E1 -3502.585,E2 -3502.585} C_VEL
LIN {X 0,Y 544.673,Z 514.652,A -85,B 0,C 180,E1 -3503.486,E2 -3503.486} C_VEL
LIN {X 0,Y 544.647,Z 510.522,A -85,B 0,C 180,E1 -3504.817,E2 -3504.817} C_VEL
LIN {X 0,Y 544.719,Z 505.869,A -85,B 0,C 180,E1 -3505.93,E2 -3505.93} C_VEL
LIN {X 0,Y 544.777,Z 498.886,A -85,B 0,C 180,E1 -3507.227,E2 -3507.227} C_VEL
LIN {X 0,Y 544.91,Z 491.35,A -85,B 0,C 180,E1 -3508.337,E2 -3508.337} C_VEL
LIN {X 0,Y 545.101,Z 481.944,A -85,B 0,C 180,E1 -3509.446,E2 -3509.446} C_VEL
LIN {X 0,Y 545.245,Z 472.301,A -85,B 0,C 180,E1 -3510.369,E2 -3510.369} C_VEL
LIN {X 0,Y 545.468,Z 461.55,A -85,B 0,C 180,E1 -3511.199,E2 -3511.199} C_VEL
LIN {X 0,Y 545.705,Z 449.323,A -85,B 0,C 180,E1 -3511.937,E2 -3511.937} C_VEL
LIN {X 0,Y 545.907,Z 437.364,A -85,B 0,C 180,E1 -3512.49,E2 -3512.49} C_VEL
LIN {X 0,Y 546.03,Z 424.998,A -85,B 0,C 180,E1 -3512.905,E2 -3512.905} C_VEL
LIN {X 0,Y 546.193,Z 412.058,A -85,B 0,C 180,E1 -3513.181,E2 -3513.181} C_VEL
LIN {X 0,Y 546.468,Z 316.506,A -85,B 0,C 180,E1 -3514.448,E2 -3514.448} C_VEL
LIN {X 0,Y 545.163,Z 308.555,A -85,B 0,C 180,E1 -3514.598,E2 -3514.598} C_VEL
LIN {X 0,Y 545.313,Z 295.206,A -85,B 0,C 180,E1 -3517.079,E2 -3517.079} C_VEL
LIN {X 0,Y 545.321,Z 284.335,A -85,B 0,C 180,E1 -3519.083,E2 -3519.083} C_VEL
LIN {X 0,Y 545.057,Z 282.592,A -85,B 0,C 180,E1 -3519.462,E2 -3519.462} C_VEL
LIN {X 0,Y 545.065,Z 282.59,A -85,B 0,C 180,E1 -3521.905,E2 -3521.905} C_VEL
LIN {X 0,Y 545.077,Z 282.583,A -85,B 0,C 180,E1 -3524.943,E2 -3524.943} C_VEL
LIN {X 0,Y 545.047,Z 282.59,A -85,B 0,C 180,E1 -3528.026,E2 -3528.026} C_VEL
LIN {X 0,Y 545.086,Z 282.589,A -85,B 0,C 180,E1 -3530.372,E2 -3530.372} C_VEL
LIN {X 0,Y 545.068,Z 282.582,A -85,B 0,C 180,E1 -3533.559,E2 -3533.559} C_VEL
LIN {X 0,Y 545.039,Z 282.593,A -85,B 0,C 180,E1 -3536.827,E2 -3536.827} C_VEL
LIN {X 0,Y 545.019,Z 282.59,A -85,B 0,C 180,E1 -3539.34,E2 -3539.34} C_VEL
LIN {X 0,Y 545.041,Z 282.586,A -85,B 0,C 180,E1 -3541.915,E2 -3541.915} C_VEL
LIN {X 0,Y 545.053,Z 282.59,A -85,B 0,C 180,E1 -3544.564,E2 -3544.564} C_VEL
LIN {X 0,Y 545.029,Z 282.591,A -85,B 0,C 180,E1 -3547.303,E2 -3547.303} C_VEL
LIN {X 0,Y 545.057,Z 282.584,A -85,B 0,C 180,E1 -3550.142,E2 -3550.142} C_VEL
LIN {X 0,Y 545.039,Z 282.596,A -85,B 0,C 180,E1 -3553.109,E2 -3553.109} C_VEL
LIN {X 0,Y 545.039,Z 282.586,A -85,B 0,C 180,E1 -3556.226,E2 -3556.226} C_VEL
LIN {X 0,Y 545.065,Z 282.588,A -85,B 0,C 180,E1 -3558.884,E2 -3558.884} C_VEL
LIN {X 0,Y 545.041,Z 282.588,A -85,B 0,C 180,E1 -3561.864,E2 -3561.864} C_VEL
LIN {X 0,Y 545.027,Z 282.588,A -85,B 0,C 180,E1 -3564.531,E2 -3564.531} C_VEL
LIN {X 0,Y 545.058,Z 282.59,A -85,B 0,C 180,E1 -3567.211,E2 -3567.211} C_VEL
LIN {X 0,Y 545.054,Z 282.59,A -85,B 0,C 180,E1 -3569.81,E2 -3569.81} C_VEL
LIN {X 0,Y 545.051,Z 282.585,A -85,B 0,C 180,E1 -3572.342,E2 -3572.342} C_VEL
LIN {X 0,Y 545.108,Z 282.578,A -85,B 0,C 180,E1 -3574.82,E2 -3574.82} C_VEL
LIN {X 0,Y 545.027,Z 282.591,A -85,B 0,C 180,E1 -3577.242,E2 -3577.242} C_VEL
LIN {X 0,Y 545.107,Z 282.579,A -85,B 0,C 180,E1 -3580.414,E2 -3580.414} C_VEL
LIN {X 0,Y 545.062,Z 282.588,A -85,B 0,C 180,E1 -3583.521,E2 -3583.521} C_VEL
LIN {X 0,Y 545.08,Z 282.59,A -85,B 0,C 180,E1 -3585.82,E2 -3585.82} C_VEL
LIN {X 0,Y 545.108,Z 282.578,A -85,B 0,C 180,E1 -3588.849,E2 -3588.849} C_VEL
LIN {X 0,Y 545.12,Z 282.582,A -85,B 0,C 180,E1 -3591.847,E2 -3591.847} C_VEL
LIN {X 0,Y 545.193,Z 282.568,A -85,B 0,C 180,E1 -3594.823,E2 -3594.823} C_VEL
LIN {X 0,Y 545.183,Z 282.571,A -85,B 0,C 180,E1 -3597.784,E2 -3597.784} C_VEL
LIN {X 0,Y 545.207,Z 282.569,A -85,B 0,C 180,E1 -3600.739,E2 -3600.739} C_VEL
LIN {X 0,Y 545.167,Z 282.572,A -85,B 0,C 180,E1 -3602.956,E2 -3602.956} C_VEL
LIN {X 0,Y 545.16,Z 282.573,A -85,B 0,C 180,E1 -3605.92,E2 -3605.92} C_VEL
LIN {X 0,Y 545.119,Z 282.581,A -85,B 0,C 180,E1 -3608.9,E2 -3608.9} C_VEL
LIN {X 0,Y 545.128,Z 282.576,A -85,B 0,C 180,E1 -3611.904,E2 -3611.904} C_VEL
LIN {X 0,Y 545.077,Z 282.588,A -85,B 0,C 180,E1 -3614.944,E2 -3614.944} C_VEL
LIN {X 0,Y 545.071,Z 282.583,A -85,B 0,C 180,E1 -3618.026,E2 -3618.026} C_VEL
LIN {X 0,Y 545.087,Z 282.583,A -85,B 0,C 180,E1 -3620.373,E2 -3620.373} C_VEL
LIN {X 0,Y 545.084,Z 282.582,A -85,B 0,C 180,E1 -3623.559,E2 -3623.559} C_VEL
LIN {X 0,Y 545.082,Z 282.581,A -85,B 0,C 180,E1 -3626.001,E2 -3626.001} C_VEL
LIN {X 0,Y 545.084,Z 282.585,A -85,B 0,C 180,E1 -3628.749,E2 -3628.749} C_VEL
LIN {X 0,Y 545.072,Z 282.585,A -85,B 0,C 180,E1 -3631.683,E2 -3631.683} C_VEL
LIN {X 0,Y 545.07,Z 282.583,A -85,B 0,C 180,E1 -3634.564,E2 -3634.564} C_VEL
LIN {X 0,Y 545.062,Z 282.594,A -85,B 0,C 180,E1 -3637.302,E2 -3637.302} C_VEL
LIN {X 0,Y 545.069,Z 282.583,A -85,B 0,C 180,E1 -3640.143,E2 -3640.143} C_VEL
LIN {X 0,Y 545.08,Z 282.586,A -85,B 0,C 180,E1 -3643.107,E2 -3643.107} C_VEL
LIN {X 0,Y 545.063,Z 282.584,A -85,B 0,C 180,E1 -3646.225,E2 -3646.225} C_VEL
LIN {X 0,Y 545.084,Z 282.581,A -85,B 0,C 180,E1 -3648.887,E2 -3648.887} C_VEL
LIN {X 0,Y 545.05,Z 282.594,A -85,B 0,C 180,E1 -3651.764,E2 -3651.764} C_VEL
LIN {X 0,Y 545.034,Z 282.587,A -85,B 0,C 180,E1 -3654.532,E2 -3654.532} C_VEL
LIN {X 0,Y 545.067,Z 282.584,A -85,B 0,C 180,E1 -3657.212,E2 -3657.212} C_VEL
LIN {X 0,Y 545.063,Z 282.592,A -85,B 0,C 180,E1 -3659.811,E2 -3659.811} C_VEL
LIN {X 0,Y 545.092,Z 282.586,A -85,B 0,C 180,E1 -3662.345,E2 -3662.345} C_VEL
LIN {X 0,Y 545.118,Z 282.581,A -85,B 0,C 180,E1 -3664.821,E2 -3664.821} C_VEL
LIN {X 0,Y 545.111,Z 282.661,A -85,B 0,C 180,E1 -3665.922,E2 -3665.922} C_VEL
LIN {X 0,Y 546.281,Z 290.052,A -85,B 0,C 180,E1 -3667.098,E2 -3667.098} C_VEL
LIN {X 0,Y 545.914,Z 310.296,A -85,B 0,C 180,E1 -3670.128,E2 -3670.128} C_VEL
LIN {X 0,Y 545.589,Z 329.493,A -85,B 0,C 180,E1 -3672.96,E2 -3672.96} C_VEL
LIN {X 0,Y 545.357,Z 346.445,A -85,B 0,C 180,E1 -3675.435,E2 -3675.435} C_VEL
LIN {X 0,Y 546.532,Z 355.372,A -85,B 0,C 180,E1 -3675.591,E2 -3675.591} C_VEL
LIN {X 0,Y 546.21,Z 454.84,A -85,B 0,C 180,E1 -3676.917,E2 -3676.917} C_VEL
LIN {X 0,Y 546.059,Z 468.127,A -85,B 0,C 180,E1 -3677.244,E2 -3677.244} C_VEL
LIN {X 0,Y 545.885,Z 480.306,A -85,B 0,C 180,E1 -3677.689,E2 -3677.689} C_VEL
LIN {X 0,Y 545.731,Z 492.635,A -85,B 0,C 180,E1 -3678.3,E2 -3678.3} C_VEL
LIN {X 0,Y 545.502,Z 504.199,A -85,B 0,C 180,E1 -3679.046,E2 -3679.046} C_VEL
LIN {X 0,Y 545.282,Z 514.611,A -85,B 0,C 180,E1 -3679.886,E2 -3679.886} C_VEL
LIN {X 0,Y 545.084,Z 523.118,A -85,B 0,C 180,E1 -3680.726,E2 -3680.726} C_VEL
LIN {X 0,Y 544.971,Z 530.965,A -85,B 0,C 180,E1 -3681.659,E2 -3681.659} C_VEL
LIN {X 0,Y 544.823,Z 538.624,A -85,B 0,C 180,E1 -3682.775,E2 -3682.775} C_VEL
LIN {X 0,Y 544.778,Z 545.682,A -85,B 0,C 180,E1 -3684.077,E2 -3684.077} C_VEL
LIN {X 0,Y 544.628,Z 550.375,A -85,B 0,C 180,E1 -3685.189,E2 -3685.189} C_VEL
LIN {X 0,Y 544.669,Z 553.959,A -85,B 0,C 180,E1 -3686.301,E2 -3686.301} C_VEL
LIN {X 0,Y 544.65,Z 555.808,A -85,B 0,C 180,E1 -3687.042,E2 -3687.042} C_VEL
LIN {X 0,Y 544.545,Z 558.183,A -85,B 0,C 180,E1 -3688.521,E2 -3688.521} C_VEL
LIN {X 0,Y 544.541,Z 559,A -85,B 0,C 180,E1 -3690,E2 -3690} C_VEL
LIN {X 0,Y 544.545,Z 558.183,A -85,B 0,C 180,E1 -3691.479,E2 -3691.479} C_VEL
LIN {X 0,Y 544.65,Z 555.809,A -85,B 0,C 180,E1 -3692.959,E2 -3692.959} C_VEL
LIN {X 0,Y 544.684,Z 552.894,A -85,B 0,C 180,E1 -3694.07,E2 -3694.07} C_VEL
LIN {X 0,Y 544.653,Z 548.947,A -85,B 0,C 180,E1 -3695.183,E2 -3695.183} C_VEL
LIN {X 0,Y 544.739,Z 543.588,A -85,B 0,C 180,E1 -3696.35,E2 -3696.35} C_VEL
LIN {X 0,Y 544.86,Z 536.233,A -85,B 0,C 180,E1 -3697.598,E2 -3697.598} C_VEL
LIN {X 0,Y 545.017,Z 527.99,A -85,B 0,C 180,E1 -3698.715,E2 -3698.715} C_VEL
LIN {X 0,Y 545.202,Z 519.537,A -85,B 0,C 180,E1 -3699.647,E2 -3699.647} C_VEL
LIN {X 0,Y 545.387,Z 509.087,A -85,B 0,C 180,E1 -3700.581,E2 -3700.581} C_VEL
LIN {X 0,Y 545.625,Z 497.375,A -85,B 0,C 180,E1 -3701.418,E2 -3701.418} C_VEL
LIN {X 0,Y 545.851,Z 485.42,A -85,B 0,C 180,E1 -3702.077,E2 -3702.077} C_VEL
LIN {X 0,Y 545.982,Z 473.057,A -85,B 0,C 180,E1 -3702.593,E2 -3702.593} C_VEL
LIN {X 0,Y 546.141,Z 460.377,A -85,B 0,C 180,E1 -3702.967,E2 -3702.967} C_VEL
LIN {X 0,Y 546.278,Z 447.14,A -85,B 0,C 180,E1 -3703.201,E2 -3703.201} C_VEL
LIN {X 0,Y 546.452,Z 353.544,A -85,B 0,C 180,E1 -3704.436,E2 -3704.436} C_VEL
LIN {X 0,Y 545.35,Z 346.459,A -85,B 0,C 180,E1 -3704.56,E2 -3704.56} C_VEL
LIN {X 0,Y 545.604,Z 325.637,A -85,B 0,C 180,E1 -3707.597,E2 -3707.597} C_VEL
LIN {X 0,Y 545.948,Z 305.72,A -85,B 0,C 180,E1 -3710.536,E2 -3710.536} C_VEL
LIN {X 0,Y 546.258,Z 289.868,A -85,B 0,C 180,E1 -3712.904,E2 -3712.904} C_VEL
LIN {X 0,Y 545.111,Z 282.588,A -85,B 0,C 180,E1 -3714.076,E2 -3714.076} C_VEL
LIN {X 0,Y 545.083,Z 282.584,A -85,B 0,C 180,E1 -3717.17,E2 -3717.17} C_VEL
LIN {X 0,Y 545.067,Z 282.587,A -85,B 0,C 180,E1 -3719.338,E2 -3719.338} C_VEL
LIN {X 0,Y 545.057,Z 282.592,A -85,B 0,C 180,E1 -3721.915,E2 -3721.915} C_VEL
LIN {X 0,Y 545.063,Z 282.59,A -85,B 0,C 180,E1 -3724.564,E2 -3724.564} C_VEL
LIN {X 0,Y 545.037,Z 282.587,A -85,B 0,C 180,E1 -3727.304,E2 -3727.304} C_VEL
LIN {X 0,Y 545.066,Z 282.589,A -85,B 0,C 180,E1 -3730.142,E2 -3730.142} C_VEL
LIN {X 0,Y 545.079,Z 282.584,A -85,B 0,C 180,E1 -3733.106,E2 -3733.106} C_VEL
LIN {X 0,Y 545.049,Z 282.589,A -85,B 0,C 180,E1 -3736.226,E2 -3736.226} C_VEL
LIN {X 0,Y 545.082,Z 282.588,A -85,B 0,C 180,E1 -3738.885,E2 -3738.885} C_VEL
LIN {X 0,Y 545.08,Z 282.591,A -85,B 0,C 180,E1 -3740.818,E2 -3740.818} C_VEL
LIN {X 0,Y 545.041,Z 282.586,A -85,B 0,C 180,E1 -3743.619,E2 -3743.619} C_VEL
LIN {X 0,Y 545.065,Z 282.583,A -85,B 0,C 180,E1 -3746.328,E2 -3746.328} C_VEL
LIN {X 0,Y 545.065,Z 282.592,A -85,B 0,C 180,E1 -3748.952,E2 -3748.952} C_VEL
LIN {X 0,Y 545.1,Z 282.583,A -85,B 0,C 180,E1 -3751.507,E2 -3751.507} C_VEL
LIN {X 0,Y 545.094,Z 282.58,A -85,B 0,C 180,E1 -3754.491,E2 -3754.491} C_VEL
LIN {X 0,Y 545.037,Z 282.595,A -85,B 0,C 180,E1 -3757.242,E2 -3757.242} C_VEL
LIN {X 0,Y 545.119,Z 282.576,A -85,B 0,C 180,E1 -3760.415,E2 -3760.415} C_VEL
LIN {X 0,Y 545.072,Z 282.592,A -85,B 0,C 180,E1 -3763.521,E2 -3763.521} C_VEL
LIN {X 0,Y 545.093,Z 282.585,A -85,B 0,C 180,E1 -3765.82,E2 -3765.82} C_VEL
LIN {X 0,Y 545.115,Z 282.576,A -85,B 0,C 180,E1 -3768.849,E2 -3768.849} C_VEL
LIN {X 0,Y 545.126,Z 282.584,A -85,B 0,C 180,E1 -3771.847,E2 -3771.847} C_VEL
LIN {X 0,Y 545.2,Z 282.564,A -85,B 0,C 180,E1 -3774.823,E2 -3774.823} C_VEL
LIN {X 0,Y 545.194,Z 282.574,A -85,B 0,C 180,E1 -3777.784,E2 -3777.784} C_VEL
LIN {X 0,Y 545.209,Z 282.565,A -85,B 0,C 180,E1 -3780.738,E2 -3780.738} C_VEL
LIN {X 0,Y 545.169,Z 282.568,A -85,B 0,C 180,E1 -3782.956,E2 -3782.956} C_VEL
LIN {X 0,Y 545.167,Z 282.575,A -85,B 0,C 180,E1 -3785.919,E2 -3785.919} C_VEL
LIN {X 0,Y 545.115,Z 282.578,A -85,B 0,C 180,E1 -3788.9,E2 -3788.9} C_VEL
LIN {X 0,Y 545.133,Z 282.577,A -85,B 0,C 180,E1 -3791.904,E2 -3791.904} C_VEL
LIN {X 0,Y 545.083,Z 282.584,A -85,B 0,C 180,E1 -3794.944,E2 -3794.944} C_VEL
LIN {X 0,Y 545.077,Z 282.583,A -85,B 0,C 180,E1 -3798.026,E2 -3798.026} C_VEL
LIN {X 0,Y 545.093,Z 282.585,A -85,B 0,C 180,E1 -3800.372,E2 -3800.372} C_VEL
LIN {X 0,Y 545.09,Z 282.58,A -85,B 0,C 180,E1 -3803.559,E2 -3803.559} C_VEL
LIN {X 0,Y 545.078,Z 282.581,A -85,B 0,C 180,E1 -3806.001,E2 -3806.001} C_VEL
LIN {X 0,Y 545.087,Z 282.587,A -85,B 0,C 180,E1 -3808.748,E2 -3808.748} C_VEL
LIN {X 0,Y 545.056,Z 282.584,A -85,B 0,C 180,E1 -3811.679,E2 -3811.679} C_VEL
LIN {X 0,Y 545.061,Z 282.585,A -85,B 0,C 180,E1 -3814.565,E2 -3814.565} C_VEL
LIN {X 0,Y 545.061,Z 282.59,A -85,B 0,C 180,E1 -3817,E2 -3817} C_VEL
LIN {X 0,Y 544.354,Z 282.679,A -85,B 0,C 180,E1 -3817.617,E2 -3817.617} C_VEL
LIN {X 0,Y 541.489,Z 283.034,A -85,B 0,C 180,E1 -3818.617,E2 -3818.617} C_VEL
LIN {X 0,Y 539.101,Z 283.333,A -85,B 0,C 180,E1 -3819.423,E2 -3819.423} C_VEL
LIN {X 0,Y 538.091,Z 283.452,A -85,B 0,C 180,E1 -3820.045,E2 -3820.045} C_VEL
LIN {X 0,Y 538.015,Z 283.46,A -85,B 0,C 180,E1 -3820.256,E2 -3820.256} C_VEL
LIN {X 0,Y 538.025,Z 283.464,A -85,B 0,C 180,E1 -3822.988,E2 -3822.988} C_VEL
LIN {X 0,Y 538.002,Z 283.464,A -85,B 0,C 180,E1 -3826.184,E2 -3826.184} C_VEL
LIN {X 0,Y 538.048,Z 283.463,A -85,B 0,C 180,E1 -3829.253,E2 -3829.253} C_VEL
LIN {X 0,Y 537.992,Z 283.468,A -85,B 0,C 180,E1 -3832.122,E2 -3832.122} C_VEL
LIN {X 0,Y 537.998,Z 283.464,A -85,B 0,C 180,E1 -3834.916,E2 -3834.916} C_VEL
LIN {X 0,Y 538.018,Z 283.47,A -85,B 0,C 180,E1 -3837.617,E2 -3837.617} C_VEL
LIN {X 0,Y 538.092,Z 283.567,A -85,B 0,C 180,E1 -3840.716,E2 -3840.716} C_VEL
LIN {X 0,Y 538.336,Z 289.239,A -85,B 0,C 180,E1 -3841.755,E2 -3841.755} C_VEL
LIN {X 0,Y 538.223,Z 305.433,A -85,B 0,C 180,E1 -3844.682,E2 -3844.682} C_VEL
LIN {X 0,Y 538.148,Z 308.642,A -85,B 0,C 180,E1 -3845.297,E2 -3845.297} C_VEL
LIN {X 0,Y 539.713,Z 318.488,A -85,B 0,C 180,E1 -3845.48,E2 -3845.48} C_VEL
LIN {X 0,Y 539.243,Z 414.98,A -85,B 0,C 180,E1 -3846.781,E2 -3846.781} C_VEL
LIN {X 0,Y 539.123,Z 428.14,A -85,B 0,C 180,E1 -3847.105,E2 -3847.105} C_VEL
LIN {X 0,Y 538.905,Z 440.918,A -85,B 0,C 180,E1 -3847.576,E2 -3847.576} C_VEL
LIN {X 0,Y 538.756,Z 453.052,A -85,B 0,C 180,E1 -3848.19,E2 -3848.19} C_VEL
LIN {X 0,Y 538.479,Z 463.492,A -85,B 0,C 180,E1 -3848.866,E2 -3848.866} C_VEL
LIN {X 0,Y 538.271,Z 474.924,A -85,B 0,C 180,E1 -3849.797,E2 -3849.797} C_VEL
LIN {X 0,Y 538.061,Z 484.256,A -85,B 0,C 180,E1 -3850.743,E2 -3850.743} C_VEL
LIN {X 0,Y 537.881,Z 493.567,A -85,B 0,C 180,E1 -3851.921,E2 -3851.921} C_VEL
LIN {X 0,Y 537.738,Z 501.049,A -85,B 0,C 180,E1 -3853.104,E2 -3853.104} C_VEL
LIN {X 0,Y 537.651,Z 505.948,A -85,B 0,C 180,E1 -3854.067,E2 -3854.067} C_VEL
LIN {X 0,Y 537.588,Z 511.086,A -85,B 0,C 180,E1 -3855.334,E2 -3855.334} C_VEL
LIN {X 0,Y 537.542,Z 514.307,A -85,B 0,C 180,E1 -3856.388,E2 -3856.388} C_VEL
LIN {X 0,Y 537.498,Z 516.102,A -85,B 0,C 180,E1 -3857.157,E2 -3857.157} C_VEL
LIN {X 0,Y 537.474,Z 517.448,A -85,B 0,C 180,E1 -3857.923,E2 -3857.923} C_VEL
LIN {X 0,Y 537.539,Z 518.389,A -85,B 0,C 180,E1 -3858.69,E2 -3858.69} C_VEL
LIN {X 0,Y 537.49,Z 518.926,A -85,B 0,C 180,E1 -3859.452,E2 -3859.452} C_VEL
LIN {X 0,Y 537.479,Z 519.02,A -85,B 0,C 180,E1 -3860.213,E2 -3860.213} C_VEL
LIN {X 0,Y 537.505,Z 518.038,A -85,B 0,C 180,E1 -3861.73,E2 -3861.73} C_VEL
LIN {X 0,Y 537.515,Z 516.952,A -85,B 0,C 180,E1 -3862.487,E2 -3862.487} C_VEL
LIN {X 0,Y 537.591,Z 514.822,A -85,B 0,C 180,E1 -3863.493,E2 -3863.493} C_VEL
LIN {X 0,Y 537.575,Z 511.11,A -85,B 0,C 180,E1 -3864.749,E2 -3864.749} C_VEL
LIN {X 0,Y 537.636,Z 506.627,A -85,B 0,C 180,E1 -3865.877,E2 -3865.877} C_VEL
LIN {X 0,Y 537.716,Z 499.851,A -85,B 0,C 180,E1 -3867.19,E2 -3867.19} C_VEL
LIN {X 0,Y 537.872,Z 492.522,A -85,B 0,C 180,E1 -3868.315,E2 -3868.315} C_VEL
LIN {X 0,Y 538.021,Z 485.075,A -85,B 0,C 180,E1 -3869.251,E2 -3869.251} C_VEL
LIN {X 0,Y 538.214,Z 476.084,A -85,B 0,C 180,E1 -3870.187,E2 -3870.187} C_VEL
LIN {X 0,Y 538.397,Z 466.15,A -85,B 0,C 180,E1 -3871.028,E2 -3871.028} C_VEL
LIN {X 0,Y 538.704,Z 455.121,A -85,B 0,C 180,E1 -3871.775,E2 -3871.775} C_VEL
LIN {X 0,Y 538.947,Z 442.804,A -85,B 0,C 180,E1 -3872.429,E2 -3872.429} C_VEL
LIN {X 0,Y 539.099,Z 430.263,A -85,B 0,C 180,E1 -3872.919,E2 -3872.919} C_VEL
LIN {X 0,Y 539.284,Z 418.014,A -85,B 0,C 180,E1 -3873.245,E2 -3873.245} C_VEL
LIN {X 0,Y 539.417,Z 397.953,A -85,B 0,C 180,E1 -3873.548,E2 -3873.548} C_VEL
LIN {X 0,Y 539.589,Z 316.927,A -85,B 0,C 180,E1 -3874.634,E2 -3874.634} C_VEL
LIN {X 0,Y 538.238,Z 308.755,A -85,B 0,C 180,E1 -3874.798,E2 -3874.798} C_VEL
LIN {X 0,Y 538.33,Z 293.173,A -85,B 0,C 180,E1 -3877.69,E2 -3877.69} C_VEL
LIN {X 0,Y 538.279,Z 285.014,A -85,B 0,C 180,E1 -3879.203,E2 -3879.203} C_VEL
LIN {X 0,Y 538.023,Z 283.469,A -85,B 0,C 180,E1 -3879.539,E2 -3879.539} C_VEL
LIN {X 0,Y 538.036,Z 283.468,A -85,B 0,C 180,E1 -3882.063,E2 -3882.063} C_VEL
LIN {X 0,Y 538.037,Z 283.459,A -85,B 0,C 180,E1 -3885.143,E2 -3885.143} C_VEL
LIN {X 0,Y 537.999,Z 283.471,A -85,B 0,C 180,E1 -3888.271,E2 -3888.271} C_VEL
LIN {X 0,Y 538.032,Z 283.466,A -85,B 0,C 180,E1 -3890.651,E2 -3890.651} C_VEL
LIN {X 0,Y 538.004,Z 283.464,A -85,B 0,C 180,E1 -3893.877,E2 -3893.877} C_VEL
LIN {X 0,Y 537.977,Z 283.472,A -85,B 0,C 180,E1 -3896.369,E2 -3896.369} C_VEL
LIN {X 0,Y 537.988,Z 283.471,A -85,B 0,C 180,E1 -3898.925,E2 -3898.925} C_VEL
LIN {X 0,Y 537.995,Z 283.464,A -85,B 0,C 180,E1 -3901.884,E2 -3901.884} C_VEL
LIN {X 0,Y 538.003,Z 283.469,A -85,B 0,C 180,E1 -3904.616,E2 -3904.616} C_VEL
LIN {X 0,Y 537.998,Z 283.469,A -85,B 0,C 180,E1 -3907.169,E2 -3907.169} C_VEL
LIN {X 0,Y 538.003,Z 283.463,A -85,B 0,C 180,E1 -3909.798,E2 -3909.798} C_VEL
LIN {X 0,Y 537.992,Z 283.473,A -85,B 0,C 180,E1 -3912.984,E2 -3912.984} C_VEL
LIN {X 0,Y 538.005,Z 283.463,A -85,B 0,C 180,E1 -3915.927,E2 -3915.927} C_VEL
LIN {X 0,Y 538.04,Z 283.468,A -85,B 0,C 180,E1 -3919.252,E2 -3919.252} C_VEL
LIN {X 0,Y 537.983,Z 283.466,A -85,B 0,C 180,E1 -3922.121,E2 -3922.121} C_VEL
LIN {X 0,Y 537.989,Z 283.467,A -85,B 0,C 180,E1 -3924.915,E2 -3924.915} C_VEL
LIN {X 0,Y 538.009,Z 283.469,A -85,B 0,C 180,E1 -3927.617,E2 -3927.617} C_VEL
LIN {X 0,Y 538.007,Z 283.463,A -85,B 0,C 180,E1 -3930.238,E2 -3930.238} C_VEL
LIN {X 0,Y 538.024,Z 283.461,A -85,B 0,C 180,E1 -3932.794,E2 -3932.794} C_VEL
LIN {X 0,Y 538.019,Z 283.465,A -85,B 0,C 180,E1 -3935.291,E2 -3935.291} C_VEL
LIN {X 0,Y 538.006,Z 283.467,A -85,B 0,C 180,E1 -3938.042,E2 -3938.042} C_VEL
LIN {X 0,Y 538.025,Z 283.46,A -85,B 0,C 180,E1 -3940.94,E2 -3940.94} C_VEL
LIN {X 0,Y 538.014,Z 283.463,A -85,B 0,C 180,E1 -3943.299,E2 -3943.299} C_VEL
LIN {X 0,Y 538.05,Z 283.462,A -85,B 0,C 180,E1 -3945.63,E2 -3945.63} C_VEL
LIN {X 0,Y 538.067,Z 283.456,A -85,B 0,C 180,E1 -3948.701,E2 -3948.701} C_VEL
LIN {X 0,Y 538.077,Z 283.458,A -85,B 0,C 180,E1 -3951.74,E2 -3951.74} C_VEL
LIN {X 0,Y 538.15,Z 283.446,A -85,B 0,C 180,E1 -3954.755,E2 -3954.755} C_VEL
LIN {X 0,Y 538.156,Z 283.446,A -85,B 0,C 180,E1 -3957.755,E2 -3957.755} C_VEL
LIN {X 0,Y 538.177,Z 283.445,A -85,B 0,C 180,E1 -3960.748,E2 -3960.748} C_VEL
LIN {X 0,Y 538.133,Z 283.448,A -85,B 0,C 180,E1 -3962.995,E2 -3962.995} C_VEL
LIN {X 0,Y 538.113,Z 283.452,A -85,B 0,C 180,E1 -3965.998,E2 -3965.998} C_VEL
LIN {X 0,Y 538.068,Z 283.458,A -85,B 0,C 180,E1 -3969.018,E2 -3969.018} C_VEL
LIN {X 0,Y 538.076,Z 283.456,A -85,B 0,C 180,E1 -3972.063,E2 -3972.063} C_VEL
LIN {X 0,Y 538.037,Z 283.462,A -85,B 0,C 180,E1 -3975.144,E2 -3975.144} C_VEL
LIN {X 0,Y 538.023,Z 283.462,A -85,B 0,C 180,E1 -3978.271,E2 -3978.271} C_VEL
LIN {X 0,Y 538.031,Z 283.466,A -85,B 0,C 180,E1 -3980.652,E2 -3980.652} C_VEL
LIN {X 0,Y 538.017,Z 283.461,A -85,B 0,C 180,E1 -3983.888,E2 -3983.888} C_VEL
LIN {X 0,Y 538.043,Z 283.459,A -85,B 0,C 180,E1 -3986.367,E2 -3986.367} C_VEL
LIN {X 0,Y 538.031,Z 283.467,A -85,B 0,C 180,E1 -3988.936,E2 -3988.936} C_VEL
LIN {X 0,Y 538.021,Z 283.461,A -85,B 0,C 180,E1 -3991.891,E2 -3991.891} C_VEL
LIN {X 0,Y 538.02,Z 283.462,A -85,B 0,C 180,E1 -3994.621,E2 -3994.621} C_VEL
LIN {X 0,Y 538.017,Z 283.469,A -85,B 0,C 180,E1 -3997.173,E2 -3997.173} C_VEL
LIN {X 0,Y 538.024,Z 283.464,A -85,B 0,C 180,E1 -3999.797,E2 -3999.797} C_VEL
LIN {X 0,Y 538.018,Z 283.462,A -85,B 0,C 180,E1 -4002.786,E2 -4002.786} C_VEL
LIN {X 0,Y 538.026,Z 283.464,A -85,B 0,C 180,E1 -4005.926,E2 -4005.926} C_VEL
LIN {X 0,Y 538.045,Z 283.462,A -85,B 0,C 180,E1 -4009.253,E2 -4009.253} C_VEL
LIN {X 0,Y 537.989,Z 283.468,A -85,B 0,C 180,E1 -4012.123,E2 -4012.123} C_VEL
LIN {X 0,Y 537.996,Z 283.464,A -85,B 0,C 180,E1 -4014.917,E2 -4014.917} C_VEL
LIN {X 0,Y 538.017,Z 283.467,A -85,B 0,C 180,E1 -4017.618,E2 -4017.618} C_VEL
LIN {X 0,Y 538.016,Z 283.468,A -85,B 0,C 180,E1 -4020.24,E2 -4020.24} C_VEL
LIN {X 0,Y 538.065,Z 283.457,A -85,B 0,C 180,E1 -4022.797,E2 -4022.797} C_VEL
LIN {X 0,Y 538.068,Z 283.538,A -85,B 0,C 180,E1 -4025.762,E2 -4025.762} C_VEL
LIN {X 0,Y 539.327,Z 291.123,A -85,B 0,C 180,E1 -4026.988,E2 -4026.988} C_VEL
LIN {X 0,Y 538.959,Z 310.057,A -85,B 0,C 180,E1 -4029.864,E2 -4029.864} C_VEL
LIN {X 0,Y 538.601,Z 329.232,A -85,B 0,C 180,E1 -4032.732,E2 -4032.732} C_VEL
LIN {X 0,Y 538.338,Z 346.167,A -85,B 0,C 180,E1 -4035.239,E2 -4035.239} C_VEL
LIN {X 0,Y 539.639,Z 355.089,A -85,B 0,C 180,E1 -4035.402,E2 -4035.402} C_VEL
LIN {X 0,Y 539.289,Z 454.555,A -85,B 0,C 180,E1 -4036.746,E2 -4036.746} C_VEL
LIN {X 0,Y 539.154,Z 467.851,A -85,B 0,C 180,E1 -4037.078,E2 -4037.078} C_VEL
LIN {X 0,Y 538.938,Z 480.032,A -85,B 0,C 180,E1 -4037.527,E2 -4037.527} C_VEL
LIN {X 0,Y 538.765,Z 491.49,A -85,B 0,C 180,E1 -4038.096,E2 -4038.096} C_VEL
LIN {X 0,Y 538.53,Z 502.646,A -85,B 0,C 180,E1 -4038.807,E2 -4038.807} C_VEL
LIN {X 0,Y 538.253,Z 513.328,A -85,B 0,C 180,E1 -4039.658,E2 -4039.658} C_VEL
LIN {X 0,Y 538.067,Z 522.957,A -85,B 0,C 180,E1 -4040.604,E2 -4040.604} C_VEL
LIN {X 0,Y 537.912,Z 530.85,A -85,B 0,C 180,E1 -4041.548,E2 -4041.548} C_VEL
LIN {X 0,Y 537.754,Z 538.56,A -85,B 0,C 180,E1 -4042.68,E2 -4042.68} C_VEL
LIN {X 0,Y 537.696,Z 545.669,A -85,B 0,C 180,E1 -4043.998,E2 -4043.998} C_VEL
LIN {X 0,Y 537.54,Z 550.375,A -85,B 0,C 180,E1 -4045.125,E2 -4045.125} C_VEL
LIN {X 0,Y 537.591,Z 553.959,A -85,B 0,C 180,E1 -4046.253,E2 -4046.253} C_VEL
LIN {X 0,Y 537.551,Z 555.807,A -85,B 0,C 180,E1 -4047.003,E2 -4047.003} C_VEL
LIN {X 0,Y 537.451,Z 558.182,A -85,B 0,C 180,E1 -4048.502,E2 -4048.502} C_VEL
LIN {X 0,Y 537.442,Z 559,A -85,B 0,C 180,E1 -4050,E2 -4050} C_VEL
LIN {X 0,Y 537.451,Z 558.183,A -85,B 0,C 180,E1 -4051.499,E2 -4051.499} C_VEL
LIN {X 0,Y 537.551,Z 555.809,A -85,B 0,C 180,E1 -4052.998,E2 -4052.998} C_VEL
LIN {X 0,Y 537.603,Z 552.894,A -85,B 0,C 180,E1 -4054.123,E2 -4054.123} C_VEL
LIN {X 0,Y 537.587,Z 548.946,A -85,B 0,C 180,E1 -4055.251,E2 -4055.251} C_VEL
LIN {X 0,Y 537.653,Z 544.053,A -85,B 0,C 180,E1 -4056.336,E2 -4056.336} C_VEL
LIN {X 0,Y 537.772,Z 537.39,A -85,B 0,C 180,E1 -4057.51,E2 -4057.51} C_VEL
LIN {X 0,Y 537.942,Z 529.349,A -85,B 0,C 180,E1 -4058.641,E2 -4058.641} C_VEL
LIN {X 0,Y 538.115,Z 521.155,A -85,B 0,C 180,E1 -4059.586,E2 -4059.586} C_VEL
LIN {X 0,Y 538.346,Z 511.165,A -85,B 0,C 180,E1 -4060.531,E2 -4060.531} C_VEL
LIN {X 0,Y 538.598,Z 501.314,A -85,B 0,C 180,E1 -4061.288,E2 -4061.288} C_VEL
LIN {X 0,Y 538.739,Z 490.106,A -85,B 0,C 180,E1 -4061.979,E2 -4061.979} C_VEL
LIN {X 0,Y 538.933,Z 477.726,A -85,B 0,C 180,E1 -4062.569,E2 -4062.569} C_VEL
LIN {X 0,Y 539.148,Z 464.666,A -85,B 0,C 180,E1 -4063.019,E2 -4063.019} C_VEL
LIN {X 0,Y 539.348,Z 451.641,A -85,B 0,C 180,E1 -4063.301,E2 -4063.301} C_VEL
LIN {X 0,Y 539.511,Z 353.66,A -85,B 0,C 180,E1 -4064.62,E2 -4064.62} C_VEL
LIN {X 0,Y 538.333,Z 346.034,A -85,B 0,C 180,E1 -4064.776,E2 -4064.776} C_VEL
LIN {X 0,Y 538.689,Z 323.652,A -85,B 0,C 180,E1 -4068.085,E2 -4068.085} C_VEL
LIN {X 0,Y 539.006,Z 305.436,A -85,B 0,C 180,E1 -4070.812,E2 -4070.812} C_VEL
LIN {X 0,Y 539.296,Z 290.896,A -85,B 0,C 180,E1 -4073.014,E2 -4073.014} C_VEL
LIN {X 0,Y 538.048,Z 283.466,A -85,B 0,C 180,E1 -4074.239,E2 -4074.239} C_VEL
LIN {X 0,Y 538.053,Z 283.461,A -85,B 0,C 180,E1 -4077.204,E2 -4077.204} C_VEL
LIN {X 0,Y 538.019,Z 283.469,A -85,B 0,C 180,E1 -4079.761,E2 -4079.761} C_VEL
LIN {X 0,Y 538.019,Z 283.468,A -85,B 0,C 180,E1 -4082.383,E2 -4082.383} C_VEL
LIN {X 0,Y 537.999,Z 283.465,A -85,B 0,C 180,E1 -4085.084,E2 -4085.084} C_VEL
LIN {X 0,Y 537.993,Z 283.468,A -85,B 0,C 180,E1 -4087.878,E2 -4087.878} C_VEL
LIN {X 0,Y 538.049,Z 283.463,A -85,B 0,C 180,E1 -4090.776,E2 -4090.776} C_VEL
LIN {X 0,Y 538.003,Z 283.464,A -85,B 0,C 180,E1 -4093.816,E2 -4093.816} C_VEL
LIN {X 0,Y 538.026,Z 283.464,A -85,B 0,C 180,E1 -4097.012,E2 -4097.012} C_VEL
LIN {X 0,Y 538.048,Z 283.459,A -85,B 0,C 180,E1 -4099.252,E2 -4099.252} C_VEL
LIN {X 0,Y 537.992,Z 283.465,A -85,B 0,C 180,E1 -4102.122,E2 -4102.122} C_VEL
LIN {X 0,Y 537.998,Z 283.473,A -85,B 0,C 180,E1 -4104.915,E2 -4104.915} C_VEL
LIN {X 0,Y 538.018,Z 283.463,A -85,B 0,C 180,E1 -4107.617,E2 -4107.617} C_VEL
LIN {X 0,Y 538.016,Z 283.461,A -85,B 0,C 180,E1 -4110.239,E2 -4110.239} C_VEL
LIN {X 0,Y 538.056,Z 283.461,A -85,B 0,C 180,E1 -4112.796,E2 -4112.796} C_VEL
LIN {X 0,Y 538.047,Z 283.467,A -85,B 0,C 180,E1 -4115.292,E2 -4115.292} C_VEL
LIN {X 0,Y 538.021,Z 283.461,A -85,B 0,C 180,E1 -4118.546,E2 -4118.546} C_VEL
LIN {X 0,Y 538.036,Z 283.461,A -85,B 0,C 180,E1 -4120.94,E2 -4120.94} C_VEL
LIN {X 0,Y 538.023,Z 283.467,A -85,B 0,C 180,E1 -4123.299,E2 -4123.299} C_VEL
LIN {X 0,Y 538.062,Z 283.463,A -85,B 0,C 180,E1 -4125.63,E2 -4125.63} C_VEL
LIN {X 0,Y 538.075,Z 283.453,A -85,B 0,C 180,E1 -4128.701,E2 -4128.701} C_VEL
LIN {X 0,Y 538.083,Z 283.461,A -85,B 0,C 180,E1 -4131.739,E2 -4131.739} C_VEL
LIN {X 0,Y 538.158,Z 283.441,A -85,B 0,C 180,E1 -4134.755,E2 -4134.755} C_VEL
LIN {X 0,Y 538.166,Z 283.449,A -85,B 0,C 180,E1 -4137.755,E2 -4137.755} C_VEL
LIN {X 0,Y 538.179,Z 283.441,A -85,B 0,C 180,E1 -4140.748,E2 -4140.748} C_VEL
LIN {X 0,Y 538.136,Z 283.444,A -85,B 0,C 180,E1 -4142.994,E2 -4142.994} C_VEL
LIN {X 0,Y 538.118,Z 283.455,A -85,B 0,C 180,E1 -4145.997,E2 -4145.997} C_VEL
LIN {X 0,Y 538.066,Z 283.455,A -85,B 0,C 180,E1 -4149.018,E2 -4149.018} C_VEL
LIN {X 0,Y 538.081,Z 283.457,A -85,B 0,C 180,E1 -4152.062,E2 -4152.062} C_VEL
LIN {X 0,Y 538.043,Z 283.459,A -85,B 0,C 180,E1 -4155.144,E2 -4155.144} C_VEL
LIN {X 0,Y 538.03,Z 283.464,A -85,B 0,C 180,E1 -4158.27,E2 -4158.27} C_VEL
LIN {X 0,Y 538.037,Z 283.467,A -85,B 0,C 180,E1 -4160.651,E2 -4160.651} C_VEL
LIN {X 0,Y 538.023,Z 283.46,A -85,B 0,C 180,E1 -4163.887,E2 -4163.887} C_VEL
LIN {X 0,Y 538.04,Z 283.461,A -85,B 0,C 180,E1 -4166.367,E2 -4166.367} C_VEL
LIN {X 0,Y 538.029,Z 283.468,A -85,B 0,C 180,E1 -4168.934,E2 -4168.934} C_VEL
LIN {X 0,Y 538.008,Z 283.461,A -85,B 0,C 180,E1 -4171.887,E2 -4171.887} C_VEL
LIN {X 0,Y 538.011,Z 283.464,A -85,B 0,C 180,E1 -4174.618,E2 -4174.618} C_VEL
LIN {X 0,Y 538.003,Z 283.472,A -85,B 0,C 180,E1 -4177.17,E2 -4177.17} C_VEL
LIN {X 0,Y 538.015,Z 283.46,A -85,B 0,C 180,E1 -4180.256,E2 -4180.256} C_VEL
LIN {X 0,Y 537.366,Z 283.546,A -85,B 0,C 180,E1 -4180.881,E2 -4180.881} C_VEL
LIN {X 0,Y 534.515,Z 283.909,A -85,B 0,C 180,E1 -4181.896,E2 -4181.896} C_VEL
LIN {X 0,Y 532.089,Z 284.214,A -85,B 0,C 180,E1 -4182.713,E2 -4182.713} C_VEL
LIN {X 0,Y 531.04,Z 284.341,A -85,B 0,C 180,E1 -4183.344,E2 -4183.344} C_VEL
LIN {X 0,Y 530.951,Z 284.349,A -85,B 0,C 180,E1 -4183.558,E2 -4183.558} C_VEL
LIN {X 0,Y 530.953,Z 284.342,A -85,B 0,C 180,E1 -4186.504,E2 -4186.504} C_VEL
LIN {X 0,Y 530.983,Z 284.34,A -85,B 0,C 180,E1 -4188.977,E2 -4188.977} C_VEL
LIN {X 0,Y 530.957,Z 284.35,A -85,B 0,C 180,E1 -4191.529,E2 -4191.529} C_VEL
LIN {X 0,Y 530.954,Z 284.343,A -85,B 0,C 180,E1 -4194.38,E2 -4194.38} C_VEL
LIN {X 0,Y 530.967,Z 284.343,A -85,B 0,C 180,E1 -4197.133,E2 -4197.133} C_VEL
LIN {X 0,Y 531.011,Z 284.343,A -85,B 0,C 180,E1 -4200.462,E2 -4200.462} C_VEL
LIN {X 0,Y 531.044,Z 284.401,A -85,B 0,C 180,E1 -4200.627,E2 -4200.627} C_VEL
LIN {X 0,Y 531.348,Z 289.514,A -85,B 0,C 180,E1 -4201.565,E2 -4201.565} C_VEL
LIN {X 0,Y 531.229,Z 305.85,A -85,B 0,C 180,E1 -4204.535,E2 -4204.535} C_VEL
LIN {X 0,Y 531.172,Z 308.786,A -85,B 0,C 180,E1 -4205.089,E2 -4205.089} C_VEL
LIN {X 0,Y 532.855,Z 319.051,A -85,B 0,C 180,E1 -4205.293,E2 -4205.293} C_VEL
LIN {X 0,Y 532.349,Z 415.762,A -85,B 0,C 180,E1 -4206.617,E2 -4206.617} C_VEL
LIN {X 0,Y 532.189,Z 429.516,A -85,B 0,C 180,E1 -4206.969,E2 -4206.969} C_VEL
LIN {X 0,Y 531.989,Z 441.425,A -85,B 0,C 180,E1 -4207.422,E2 -4207.422} C_VEL
LIN {X 0,Y 531.822,Z 453.372,A -85,B 0,C 180,E1 -4208.037,E2 -4208.037} C_VEL
LIN {X 0,Y 531.518,Z 464.568,A -85,B 0,C 180,E1 -4208.779,E2 -4208.779} C_VEL
LIN {X 0,Y 531.289,Z 475.412,A -85,B 0,C 180,E1 -4209.681,E2 -4209.681} C_VEL
LIN {X 0,Y 531.028,Z 485.025,A -85,B 0,C 180,E1 -4210.678,E2 -4210.678} C_VEL
LIN {X 0,Y 530.828,Z 494.25,A -85,B 0,C 180,E1 -4211.872,E2 -4211.872} C_VEL
LIN {X 0,Y 530.687,Z 501.584,A -85,B 0,C 180,E1 -4213.061,E2 -4213.061} C_VEL
LIN {X 0,Y 530.56,Z 507.349,A -85,B 0,C 180,E1 -4214.243,E2 -4214.243} C_VEL
LIN {X 0,Y 530.509,Z 511.839,A -85,B 0,C 180,E1 -4215.421,E2 -4215.421} C_VEL
LIN {X 0,Y 530.471,Z 514.194,A -85,B 0,C 180,E1 -4216.203,E2 -4216.203} C_VEL
LIN {X 0,Y 530.411,Z 516.098,A -85,B 0,C 180,E1 -4216.982,E2 -4216.982} C_VEL
LIN {X 0,Y 530.388,Z 517.515,A -85,B 0,C 180,E1 -4217.76,E2 -4217.76} C_VEL
LIN {X 0,Y 530.448,Z 518.63,A -85,B 0,C 180,E1 -4218.649,E2 -4218.649} C_VEL
LIN {X 0,Y 530.389,Z 519.311,A -85,B 0,C 180,E1 -4220.081,E2 -4220.081} C_VEL
LIN {X 0,Y 530.415,Z 518.442,A -85,B 0,C 180,E1 -4221.619,E2 -4221.619} C_VEL
LIN {X 0,Y 530.425,Z 517.426,A -85,B 0,C 180,E1 -4222.386,E2 -4222.386} C_VEL
LIN {X 0,Y 530.524,Z 515.205,A -85,B 0,C 180,E1 -4223.487,E2 -4223.487} C_VEL
LIN {X 0,Y 530.505,Z 511.802,A -85,B 0,C 180,E1 -4224.679,E2 -4224.679} C_VEL
LIN {X 0,Y 530.553,Z 507.449,A -85,B 0,C 180,E1 -4225.822,E2 -4225.822} C_VEL
LIN {X 0,Y 530.599,Z 501.931,A -85,B 0,C 180,E1 -4226.963,E2 -4226.963} C_VEL
LIN {X 0,Y 530.768,Z 495.05,A -85,B 0,C 180,E1 -4228.103,E2 -4228.103} C_VEL
LIN {X 0,Y 530.979,Z 486.453,A -85,B 0,C 180,E1 -4229.241,E2 -4229.241} C_VEL
LIN {X 0,Y 531.196,Z 477.68,A -85,B 0,C 180,E1 -4230.189,E2 -4230.189} C_VEL
LIN {X 0,Y 531.363,Z 468.082,A -85,B 0,C 180,E1 -4231.042,E2 -4231.042} C_VEL
LIN {X 0,Y 531.714,Z 457.529,A -85,B 0,C 180,E1 -4231.798,E2 -4231.798} C_VEL
LIN {X 0,Y 531.959,Z 445.779,A -85,B 0,C 180,E1 -4232.46,E2 -4232.46} C_VEL
LIN {X 0,Y 532.149,Z 433.603,A -85,B 0,C 180,E1 -4232.98,E2 -4232.98} C_VEL
LIN {X 0,Y 532.342,Z 421.961,A -85,B 0,C 180,E1 -4233.334,E2 -4233.334} C_VEL
LIN {X 0,Y 532.458,Z 409.721,A -85,B 0,C 180,E1 -4233.57,E2 -4233.57} C_VEL
LIN {X 0,Y 532.67,Z 317.413,A -85,B 0,C 180,E1 -4234.824,E2 -4234.824} C_VEL
LIN {X 0,Y 531.246,Z 308.909,A -85,B 0,C 180,E1 -4235.004,E2 -4235.004} C_VEL
LIN {X 0,Y 531.355,Z 292.917,A -85,B 0,C 180,E1 -4237.982,E2 -4237.982} C_VEL
LIN {X 0,Y 531.203,Z 285.752,A -85,B 0,C 180,E1 -4239.327,E2 -4239.327} C_VEL
LIN {X 0,Y 530.991,Z 284.345,A -85,B 0,C 180,E1 -4239.619,E2 -4239.619} C_VEL
LIN {X 0,Y 531.007,Z 284.345,A -85,B 0,C 180,E1 -4242.225,E2 -4242.225} C_VEL
LIN {X 0,Y 530.983,Z 284.337,A -85,B 0,C 180,E1 -4245.349,E2 -4245.349} C_VEL
LIN {X 0,Y 530.956,Z 284.349,A -85,B 0,C 180,E1 -4248.522,E2 -4248.522} C_VEL
LIN {X 0,Y 530.995,Z 284.339,A -85,B 0,C 180,E1 -4250.937,E2 -4250.937} C_VEL
LIN {X 0,Y 530.946,Z 284.347,A -85,B 0,C 180,E1 -4254.225,E2 -4254.225} C_VEL
LIN {X 0,Y 530.944,Z 284.35,A -85,B 0,C 180,E1 -4256.746,E2 -4256.746} C_VEL
LIN {X 0,Y 530.957,Z 284.342,A -85,B 0,C 180,E1 -4259.323,E2 -4259.323} C_VEL
LIN {X 0,Y 530.952,Z 284.342,A -85,B 0,C 180,E1 -4262.098,E2 -4262.098} C_VEL
LIN {X 0,Y 530.963,Z 284.35,A -85,B 0,C 180,E1 -4264.85,E2 -4264.85} C_VEL
LIN {X 0,Y 530.959,Z 284.342,A -85,B 0,C 180,E1 -4267.507,E2 -4267.507} C_VEL
LIN {X 0,Y 530.945,Z 284.344,A -85,B 0,C 180,E1 -4270.435,E2 -4270.435} C_VEL
LIN {X 0,Y 530.938,Z 284.346,A -85,B 0,C 180,E1 -4273.496,E2 -4273.496} C_VEL
LIN {X 0,Y 530.931,Z 284.345,A -85,B 0,C 180,E1 -4276.502,E2 -4276.502} C_VEL
LIN {X 0,Y 530.969,Z 284.344,A -85,B 0,C 180,E1 -4279.566,E2 -4279.566} C_VEL
LIN {X 0,Y 530.96,Z 284.341,A -85,B 0,C 180,E1 -4282.577,E2 -4282.577} C_VEL
LIN {X 0,Y 530.974,Z 284.347,A -85,B 0,C 180,E1 -4285.309,E2 -4285.309} C_VEL
LIN {X 0,Y 530.958,Z 284.342,A -85,B 0,C 180,E1 -4288.031,E2 -4288.031} C_VEL
LIN {X 0,Y 530.98,Z 284.339,A -85,B 0,C 180,E1 -4290.874,E2 -4290.874} C_VEL
LIN {X 0,Y 530.98,Z 284.342,A -85,B 0,C 180,E1 -4293.255,E2 -4293.255} C_VEL
LIN {X 0,Y 530.95,Z 284.347,A -85,B 0,C 180,E1 -4295.967,E2 -4295.967} C_VEL
LIN {X 0,Y 530.989,Z 284.337,A -85,B 0,C 180,E1 -4299.062,E2 -4299.062} C_VEL
LIN {X 0,Y 530.98,Z 284.342,A -85,B 0,C 180,E1 -4301.478,E2 -4301.478} C_VEL
LIN {X 0,Y 530.984,Z 284.338,A -85,B 0,C 180,E1 -4304.65,E2 -4304.65} C_VEL
LIN {X 0,Y 531.03,Z 284.338,A -85,B 0,C 180,E1 -4307.775,E2 -4307.775} C_VEL
LIN {X 0,Y 531.02,Z 284.333,A -85,B 0,C 180,E1 -4310.862,E2 -4310.862} C_VEL
LIN {X 0,Y 531.006,Z 284.334,A -85,B 0,C 180,E1 -4313.159,E2 -4313.159} C_VEL
LIN {X 0,Y 531.109,Z 284.324,A -85,B 0,C 180,E1 -4314.685,E2 -4314.685} C_VEL
LIN {X 0,Y 531.128,Z 284.322,A -85,B 0,C 180,E1 -4317.725,E2 -4317.725} C_VEL
LIN {X 0,Y 531.146,Z 284.32,A -85,B 0,C 180,E1 -4320.758,E2 -4320.758} C_VEL
LIN {X 0,Y 531.099,Z 284.324,A -85,B 0,C 180,E1 -4323.034,E2 -4323.034} C_VEL
LIN {X 0,Y 531.073,Z 284.33,A -85,B 0,C 180,E1 -4326.077,E2 -4326.077} C_VEL
LIN {X 0,Y 531.027,Z 284.334,A -85,B 0,C 180,E1 -4329.138,E2 -4329.138} C_VEL
LIN {X 0,Y 531.033,Z 284.335,A -85,B 0,C 180,E1 -4332.225,E2 -4332.225} C_VEL
LIN {X 0,Y 530.987,Z 284.338,A -85,B 0,C 180,E1 -4335.35,E2 -4335.35} C_VEL
LIN {X 0,Y 530.983,Z 284.343,A -85,B 0,C 180,E1 -4338.522,E2 -4338.522} C_VEL
LIN {X 0,Y 530.992,Z 284.345,A -85,B 0,C 180,E1 -4340.938,E2 -4340.938} C_VEL
LIN {X 0,Y 530.973,Z 284.339,A -85,B 0,C 180,E1 -4344.225,E2 -4344.225} C_VEL
LIN {X 0,Y 531.004,Z 284.34,A -85,B 0,C 180,E1 -4346.744,E2 -4346.744} C_VEL
LIN {X 0,Y 530.987,Z 284.343,A -85,B 0,C 180,E1 -4349.323,E2 -4349.323} C_VEL
LIN {X 0,Y 530.974,Z 284.338,A -85,B 0,C 180,E1 -4352.104,E2 -4352.104} C_VEL
LIN {X 0,Y 530.977,Z 284.342,A -85,B 0,C 180,E1 -4354.854,E2 -4354.854} C_VEL
LIN {X 0,Y 530.967,Z 284.346,A -85,B 0,C 180,E1 -4357.508,E2 -4357.508} C_VEL
LIN {X 0,Y 530.98,Z 284.338,A -85,B 0,C 180,E1 -4360.433,E2 -4360.433} C_VEL
LIN {X 0,Y 530.964,Z 284.347,A -85,B 0,C 180,E1 -4363.283,E2 -4363.283} C_VEL
LIN {X 0,Y 530.984,Z 284.346,A -85,B 0,C 180,E1 -4365.622,E2 -4365.622} C_VEL
LIN {X 0,Y 530.994,Z 284.336,A -85,B 0,C 180,E1 -4368.566,E2 -4368.566} C_VEL
LIN {X 0,Y 530.954,Z 284.348,A -85,B 0,C 180,E1 -4371.53,E2 -4371.53} C_VEL
LIN {X 0,Y 530.952,Z 284.343,A -85,B 0,C 180,E1 -4374.381,E2 -4374.381} C_VEL
LIN {X 0,Y 530.965,Z 284.34,A -85,B 0,C 180,E1 -4377.134,E2 -4377.134} C_VEL
LIN {X 0,Y 530.969,Z 284.347,A -85,B 0,C 180,E1 -4379.804,E2 -4379.804} C_VEL
LIN {X 0,Y 531.015,Z 284.338,A -85,B 0,C 180,E1 -4382.468,E2 -4382.468} C_VEL
LIN {X 0,Y 531.034,Z 284.401,A -85,B 0,C 180,E1 -4385.597,E2 -4385.597} C_VEL
LIN {X 0,Y 532.376,Z 292.185,A -85,B 0,C 180,E1 -4386.876,E2 -4386.876} C_VEL
LIN {X 0,Y 531.994,Z 310.599,A -85,B 0,C 180,E1 -4389.712,E2 -4389.712} C_VEL
LIN {X 0,Y 531.583,Z 330.276,A -85,B 0,C 180,E1 -4392.695,E2 -4392.695} C_VEL
LIN {X 0,Y 531.307,Z 345.951,A -85,B 0,C 180,E1 -4395.046,E2 -4395.046} C_VEL
LIN {X 0,Y 532.759,Z 355.533,A -85,B 0,C 180,E1 -4395.219,E2 -4395.219} C_VEL
LIN {X 0,Y 532.384,Z 454.271,A -85,B 0,C 180,E1 -4396.571,E2 -4396.571} C_VEL
LIN {X 0,Y 532.228,Z 467.574,A -85,B 0,C 180,E1 -4396.907,E2 -4396.907} C_VEL
LIN {X 0,Y 531.974,Z 479.758,A -85,B 0,C 180,E1 -4397.361,E2 -4397.361} C_VEL
LIN {X 0,Y 531.763,Z 491.697,A -85,B 0,C 180,E1 -4397.964,E2 -4397.964} C_VEL
LIN {X 0,Y 531.5,Z 503.674,A -85,B 0,C 180,E1 -4398.754,E2 -4398.754} C_VEL
LIN {X 0,Y 531.203,Z 514.134,A -85,B 0,C 180,E1 -4399.615,E2 -4399.615} C_VEL
LIN {X 0,Y 531.018,Z 522.689,A -85,B 0,C 180,E1 -4400.478,E2 -4400.478} C_VEL
LIN {X 0,Y 530.868,Z 530.584,A -85,B 0,C 180,E1 -4401.435,E2 -4401.435} C_VEL
LIN {X 0,Y 530.674,Z 538.294,A -85,B 0,C 180,E1 -4402.582,E2 -4402.582} C_VEL
LIN {X 0,Y 530.588,Z 545.404,A -85,B 0,C 180,E1 -4403.918,E2 -4403.918} C_VEL
LIN {X 0,Y 530.459,Z 550.131,A -85,B 0,C 180,E1 -4405.06,E2 -4405.06} C_VEL
LIN {X 0,Y 530.516,Z 553.747,A -85,B 0,C 180,E1 -4406.203,E2 -4406.203} C_VEL
LIN {X 0,Y 530.457,Z 555.609,A -85,B 0,C 180,E1 -4406.963,E2 -4406.963} C_VEL
LIN {X 0,Y 530.41,Z 557.006,A -85,B 0,C 180,E1 -4407.722,E2 -4407.722} C_VEL
LIN {X 0,Y 530.344,Z 558.609,A -85,B 0,C 180,E1 -4409.241,E2 -4409.241} C_VEL
LIN {X 0,Y 530.345,Z 558.826,A -85,B 0,C 180,E1 -4410,E2 -4410} C_VEL
LIN {X 0,Y 530.361,Z 558.001,A -85,B 0,C 180,E1 -4411.519,E2 -4411.519} C_VEL
LIN {X 0,Y 530.41,Z 557.006,A -85,B 0,C 180,E1 -4412.278,E2 -4412.278} C_VEL
LIN {X 0,Y 530.457,Z 555.61,A -85,B 0,C 180,E1 -4413.038,E2 -4413.038} C_VEL
LIN {X 0,Y 530.522,Z 552.671,A -85,B 0,C 180,E1 -4414.179,E2 -4414.179} C_VEL
LIN {X 0,Y 530.525,Z 548.689,A -85,B 0,C 180,E1 -4415.321,E2 -4415.321} C_VEL
LIN {X 0,Y 530.566,Z 543.125,A -85,B 0,C 180,E1 -4416.551,E2 -4416.551} C_VEL
LIN {X 0,Y 530.73,Z 535.88,A -85,B 0,C 180,E1 -4417.801,E2 -4417.801} C_VEL
LIN {X 0,Y 530.911,Z 527.581,A -85,B 0,C 180,E1 -4418.949,E2 -4418.949} C_VEL
LIN {X 0,Y 531.105,Z 519.076,A -85,B 0,C 180,E1 -4419.906,E2 -4419.906} C_VEL
LIN {X 0,Y 531.359,Z 508.569,A -85,B 0,C 180,E1 -4420.864,E2 -4420.864} C_VEL
LIN {X 0,Y 531.627,Z 497.59,A -85,B 0,C 180,E1 -4421.671,E2 -4421.671} C_VEL
LIN {X 0,Y 531.876,Z 486.785,A -85,B 0,C 180,E1 -4422.303,E2 -4422.303} C_VEL
LIN {X 0,Y 532.065,Z 475.095,A -85,B 0,C 180,E1 -4422.831,E2 -4422.831} C_VEL
LIN {X 0,Y 532.284,Z 461.629,A -85,B 0,C 180,E1 -4423.263,E2 -4423.263} C_VEL
LIN {X 0,Y 532.463,Z 448.309,A -85,B 0,C 180,E1 -4423.525,E2 -4423.525} C_VEL
LIN {X 0,Y 532.673,Z 354.669,A -85,B 0,C 180,E1 -4424.795,E2 -4424.795} C_VEL
LIN {X 0,Y 531.305,Z 345.844,A -85,B 0,C 180,E1 -4424.963,E2 -4424.963} C_VEL
LIN {X 0,Y 531.712,Z 323.559,A -85,B 0,C 180,E1 -4428.303,E2 -4428.303} C_VEL
LIN {X 0,Y 532.082,Z 303.827,A -85,B 0,C 180,E1 -4431.299,E2 -4431.299} C_VEL
LIN {X 0,Y 532.339,Z 291.929,A -85,B 0,C 180,E1 -4433.127,E2 -4433.127} C_VEL
LIN {X 0,Y 531.017,Z 284.34,A -85,B 0,C 180,E1 -4434.379,E2 -4434.379} C_VEL
LIN {X 0,Y 531,Z 284.34,A -85,B 0,C 180,E1 -4436.744,E2 -4436.744} C_VEL
LIN {X 0,Y 530.984,Z 284.342,A -85,B 0,C 180,E1 -4439.322,E2 -4439.322} C_VEL
LIN {X 0,Y 530.967,Z 284.351,A -85,B 0,C 180,E1 -4442.1,E2 -4442.1} C_VEL
LIN {X 0,Y 530.971,Z 284.342,A -85,B 0,C 180,E1 -4444.851,E2 -4444.851} C_VEL
LIN {X 0,Y 530.967,Z 284.341,A -85,B 0,C 180,E1 -4447.507,E2 -4447.507} C_VEL
LIN {X 0,Y 530.982,Z 284.347,A -85,B 0,C 180,E1 -4450.433,E2 -4450.433} C_VEL
LIN {X 0,Y 530.961,Z 284.342,A -85,B 0,C 180,E1 -4453.281,E2 -4453.281} C_VEL
LIN {X 0,Y 530.976,Z 284.339,A -85,B 0,C 180,E1 -4455.622,E2 -4455.622} C_VEL
LIN {X 0,Y 530.993,Z 284.344,A -85,B 0,C 180,E1 -4458.564,E2 -4458.564} C_VEL
LIN {X 0,Y 530.957,Z 284.342,A -85,B 0,C 180,E1 -4461.529,E2 -4461.529} C_VEL
LIN {X 0,Y 530.954,Z 284.343,A -85,B 0,C 180,E1 -4464.38,E2 -4464.38} C_VEL
LIN {X 0,Y 530.966,Z 284.347,A -85,B 0,C 180,E1 -4467.133,E2 -4467.133} C_VEL
LIN {X 0,Y 530.968,Z 284.339,A -85,B 0,C 180,E1 -4469.803,E2 -4469.803} C_VEL
LIN {X 0,Y 531.011,Z 284.335,A -85,B 0,C 180,E1 -4472.467,E2 -4472.467} C_VEL
LIN {X 0,Y 531.004,Z 284.34,A -85,B 0,C 180,E1 -4474.942,E2 -4474.942} C_VEL
LIN {X 0,Y 530.97,Z 284.339,A -85,B 0,C 180,E1 -4478.246,E2 -4478.246} C_VEL
LIN {X 0,Y 530.994,Z 284.336,A -85,B 0,C 180,E1 -4480.677,E2 -4480.677} C_VEL
LIN {X 0,Y 530.984,Z 284.34,A -85,B 0,C 180,E1 -4483.071,E2 -4483.071} C_VEL
LIN {X 0,Y 531.039,Z 284.338,A -85,B 0,C 180,E1 -4485.436,E2 -4485.436} C_VEL
LIN {X 0,Y 531.034,Z 284.33,A -85,B 0,C 180,E1 -4488.55,E2 -4488.55} C_VEL
LIN {X 0,Y 531.053,Z 284.335,A -85,B 0,C 180,E1 -4491.629,E2 -4491.629} C_VEL
LIN {X 0,Y 531.117,Z 284.318,A -85,B 0,C 180,E1 -4494.685,E2 -4494.685} C_VEL
LIN {X 0,Y 531.138,Z 284.324,A -85,B 0,C 180,E1 -4497.725,E2 -4497.725} C_VEL
LIN {X 0,Y 531.15,Z 284.316,A -85,B 0,C 180,E1 -4500.758,E2 -4500.758} C_VEL
LIN {X 0,Y 531.103,Z 284.32,A -85,B 0,C 180,E1 -4503.034,E2 -4503.034} C_VEL
LIN {X 0,Y 531.074,Z 284.333,A -85,B 0,C 180,E1 -4506.077,E2 -4506.077} C_VEL
LIN {X 0,Y 531.053,Z 284.336,A -85,B 0,C 180,E1 -4508.37,E2 -4508.37} C_VEL
LIN {X 0,Y 531.049,Z 284.329,A -85,B 0,C 180,E1 -4511.672,E2 -4511.672} C_VEL
LIN {X 0,Y 531.029,Z 284.334,A -85,B 0,C 180,E1 -4514.956,E2 -4514.956} C_VEL
LIN {X 0,Y 531.015,Z 284.333,A -85,B 0,C 180,E1 -4517.722,E2 -4517.722} C_VEL
LIN {X 0,Y 530.998,Z 284.341,A -85,B 0,C 180,E1 -4520.938,E2 -4520.938} C_VEL
LIN {X 0,Y 530.979,Z 284.34,A -85,B 0,C 180,E1 -4524.225,E2 -4524.225} C_VEL
LIN {X 0,Y 531,Z 284.343,A -85,B 0,C 180,E1 -4526.744,E2 -4526.744} C_VEL
LIN {X 0,Y 530.98,Z 284.341,A -85,B 0,C 180,E1 -4529.323,E2 -4529.323} C_VEL
LIN {X 0,Y 530.964,Z 284.338,A -85,B 0,C 180,E1 -4532.1,E2 -4532.1} C_VEL
LIN {X 0,Y 530.969,Z 284.344,A -85,B 0,C 180,E1 -4534.851,E2 -4534.851} C_VEL
LIN {X 0,Y 530.964,Z 284.345,A -85,B 0,C 180,E1 -4537.508,E2 -4537.508} C_VEL
LIN {X 0,Y 530.98,Z 284.337,A -85,B 0,C 180,E1 -4540.433,E2 -4540.433} C_VEL
LIN {X 0,Y 530.96,Z 284.349,A -85,B 0,C 180,E1 -4543.281,E2 -4543.281} C_VEL
LIN {X 0,Y 530.951,Z 284.349,A -85,B 0,C 180,E1 -4543.558,E2 -4543.558} C_VEL
LIN {X 0,Y 530.277,Z 284.429,A -85,B 0,C 180,E1 -4544.191,E2 -4544.191} C_VEL
LIN {X 0,Y 527.43,Z 284.787,A -85,B 0,C 180,E1 -4545.22,E2 -4545.22} C_VEL
LIN {X 0,Y 525.029,Z 285.082,A -85,B 0,C 180,E1 -4546.049,E2 -4546.049} C_VEL
LIN {X 0,Y 523.998,Z 285.209,A -85,B 0,C 180,E1 -4546.688,E2 -4546.688} C_VEL
LIN {X 0,Y 523.914,Z 285.22,A -85,B 0,C 180,E1 -4546.905,E2 -4546.905} C_VEL
LIN {X 0,Y 523.948,Z 285.22,A -85,B 0,C 180,E1 -4549.921,E2 -4549.921} C_VEL
LIN {X 0,Y 523.907,Z 285.22,A -85,B 0,C 180,E1 -4552.868,E2 -4552.868} C_VEL
LIN {X 0,Y 523.933,Z 285.226,A -85,B 0,C 180,E1 -4555.71,E2 -4555.71} C_VEL
LIN {X 0,Y 523.921,Z 285.223,A -85,B 0,C 180,E1 -4558.456,E2 -4558.456} C_VEL
LIN {X 0,Y 523.978,Z 285.263,A -85,B 0,C 180,E1 -4560.527,E2 -4560.527} C_VEL
LIN {X 0,Y 524.345,Z 289.775,A -85,B 0,C 180,E1 -4561.369,E2 -4561.369} C_VEL
LIN {X 0,Y 524.227,Z 305.663,A -85,B 0,C 180,E1 -4564.264,E2 -4564.264} C_VEL
LIN {X 0,Y 524.189,Z 309.056,A -85,B 0,C 180,E1 -4564.886,E2 -4564.886} C_VEL
LIN {X 0,Y 526.008,Z 320.344,A -85,B 0,C 180,E1 -4565.111,E2 -4565.111} C_VEL
LIN {X 0,Y 525.46,Z 415.24,A -85,B 0,C 180,E1 -4566.422,E2 -4566.422} C_VEL
LIN {X 0,Y 525.322,Z 428.517,A -85,B 0,C 180,E1 -4566.755,E2 -4566.755} C_VEL
LIN {X 0,Y 525.121,Z 440.775,A -85,B 0,C 180,E1 -4567.215,E2 -4567.215} C_VEL
LIN {X 0,Y 524.886,Z 453.17,A -85,B 0,C 180,E1 -4567.847,E2 -4567.847} C_VEL
LIN {X 0,Y 524.585,Z 464.299,A -85,B 0,C 180,E1 -4568.588,E2 -4568.588} C_VEL
LIN {X 0,Y 524.309,Z 475.232,A -85,B 0,C 180,E1 -4569.501,E2 -4569.501} C_VEL
LIN {X 0,Y 524.063,Z 484.078,A -85,B 0,C 180,E1 -4570.411,E2 -4570.411} C_VEL
LIN {X 0,Y 523.876,Z 492.141,A -85,B 0,C 180,E1 -4571.421,E2 -4571.421} C_VEL
LIN {X 0,Y 523.671,Z 499.625,A -85,B 0,C 180,E1 -4572.574,E2 -4572.574} C_VEL
LIN {X 0,Y 523.513,Z 505.18,A -85,B 0,C 180,E1 -4573.625,E2 -4573.625} C_VEL
LIN {X 0,Y 523.475,Z 510.375,A -85,B 0,C 180,E1 -4574.863,E2 -4574.863} C_VEL
LIN {X 0,Y 523.41,Z 514.08,A -85,B 0,C 180,E1 -4576.013,E2 -4576.013} C_VEL
LIN {X 0,Y 523.327,Z 516.049,A -85,B 0,C 180,E1 -4576.803,E2 -4576.803} C_VEL
LIN {X 0,Y 523.296,Z 517.578,A -85,B 0,C 180,E1 -4577.591,E2 -4577.591} C_VEL
LIN {X 0,Y 523.363,Z 518.867,A -85,B 0,C 180,E1 -4578.604,E2 -4578.604} C_VEL
LIN {X 0,Y 523.308,Z 519.563,A -85,B 0,C 180,E1 -4579.945,E2 -4579.945} C_VEL
LIN {X 0,Y 523.269,Z 519.42,A -85,B 0,C 180,E1 -4580.725,E2 -4580.725} C_VEL
LIN {X 0,Y 523.32,Z 518.846,A -85,B 0,C 180,E1 -4581.505,E2 -4581.505} C_VEL
LIN {X 0,Y 523.353,Z 517.885,A -85,B 0,C 180,E1 -4582.282,E2 -4582.282} C_VEL
LIN {X 0,Y 523.457,Z 515.588,A -85,B 0,C 180,E1 -4583.481,E2 -4583.481} C_VEL
LIN {X 0,Y 523.437,Z 512.493,A -85,B 0,C 180,E1 -4584.607,E2 -4584.607} C_VEL
LIN {X 0,Y 523.475,Z 508.269,A -85,B 0,C 180,E1 -4585.765,E2 -4585.765} C_VEL
LIN {X 0,Y 523.589,Z 501.886,A -85,B 0,C 180,E1 -4587.114,E2 -4587.114} C_VEL
LIN {X 0,Y 523.736,Z 494.912,A -85,B 0,C 180,E1 -4588.269,E2 -4588.269} C_VEL
LIN {X 0,Y 523.983,Z 486.227,A -85,B 0,C 180,E1 -4589.423,E2 -4589.423} C_VEL
LIN {X 0,Y 524.195,Z 477.363,A -85,B 0,C 180,E1 -4590.384,E2 -4590.384} C_VEL
LIN {X 0,Y 524.445,Z 467.631,A -85,B 0,C 180,E1 -4591.247,E2 -4591.247} C_VEL
LIN {X 0,Y 524.8,Z 456.85,A -85,B 0,C 180,E1 -4592.014,E2 -4592.014} C_VEL
LIN {X 0,Y 525.081,Z 444.838,A -85,B 0,C 180,E1 -4592.685,E2 -4592.685} C_VEL
LIN {X 0,Y 525.274,Z 432.297,A -85,B 0,C 180,E1 -4593.211,E2 -4593.211} C_VEL
LIN {X 0,Y 525.459,Z 420.887,A -85,B 0,C 180,E1 -4593.546,E2 -4593.546} C_VEL
LIN {X 0,Y 525.563,Z 405.745,A -85,B 0,C 180,E1 -4593.809,E2 -4593.809} C_VEL
LIN {X 0,Y 525.851,Z 318.417,A -85,B 0,C 180,E1 -4595.01,E2 -4595.01} C_VEL
LIN {X 0,Y 524.23,Z 309.191,A -85,B 0,C 180,E1 -4595.191,E2 -4595.191} C_VEL
LIN {X 0,Y 524.373,Z 293.724,A -85,B 0,C 180,E1 -4598.089,E2 -4598.089} C_VEL
LIN {X 0,Y 524.309,Z 287.498,A -85,B 0,C 180,E1 -4599.256,E2 -4599.256} C_VEL
LIN {X 0,Y 523.958,Z 285.222,A -85,B 0,C 180,E1 -4599.749,E2 -4599.749} C_VEL
LIN {X 0,Y 523.945,Z 285.223,A -85,B 0,C 180,E1 -4602.393,E2 -4602.393} C_VEL
LIN {X 0,Y 523.921,Z 285.217,A -85,B 0,C 180,E1 -4605.562,E2 -4605.562} C_VEL
LIN {X 0,Y 523.91,Z 285.222,A -85,B 0,C 180,E1 -4607.97,E2 -4607.97} C_VEL
LIN {X 0,Y 523.951,Z 285.223,A -85,B 0,C 180,E1 -4610.41,E2 -4610.41} C_VEL
LIN {X 0,Y 523.906,Z 285.223,A -85,B 0,C 180,E1 -4612.893,E2 -4612.893} C_VEL
LIN {X 0,Y 523.891,Z 285.221,A -85,B 0,C 180,E1 -4615.421,E2 -4615.421} C_VEL
LIN {X 0,Y 523.902,Z 285.221,A -85,B 0,C 180,E1 -4618.002,E2 -4618.002} C_VEL
LIN {X 0,Y 523.904,Z 285.227,A -85,B 0,C 180,E1 -4620.847,E2 -4620.847} C_VEL
LIN {X 0,Y 523.925,Z 285.217,A -85,B 0,C 180,E1 -4623.729,E2 -4623.729} C_VEL
LIN {X 0,Y 523.898,Z 285.223,A -85,B 0,C 180,E1 -4626.4,E2 -4626.4} C_VEL
LIN {X 0,Y 523.907,Z 285.227,A -85,B 0,C 180,E1 -4629.085,E2 -4629.085} C_VEL
LIN {X 0,Y 523.905,Z 285.219,A -85,B 0,C 180,E1 -4632.122,E2 -4632.122} C_VEL
LIN {X 0,Y 523.932,Z 285.222,A -85,B 0,C 180,E1 -4635.31,E2 -4635.31} C_VEL
LIN {X 0,Y 523.944,Z 285.217,A -85,B 0,C 180,E1 -4638.69,E2 -4638.69} C_VEL
LIN {X 0,Y 523.907,Z 285.22,A -85,B 0,C 180,E1 -4641.897,E2 -4641.897} C_VEL
LIN {X 0,Y 523.916,Z 285.221,A -85,B 0,C 180,E1 -4644.911,E2 -4644.911} C_VEL
LIN {X 0,Y 523.927,Z 285.223,A -85,B 0,C 180,E1 -4647.679,E2 -4647.679} C_VEL
LIN {X 0,Y 523.945,Z 285.214,A -85,B 0,C 180,E1 -4650.676,E2 -4650.676} C_VEL
LIN {X 0,Y 523.96,Z 285.22,A -85,B 0,C 180,E1 -4653.728,E2 -4653.728} C_VEL
LIN {X 0,Y 523.903,Z 285.221,A -85,B 0,C 180,E1 -4656.269,E2 -4656.269} C_VEL
LIN {X 0,Y 523.936,Z 285.215,A -85,B 0,C 180,E1 -4658.766,E2 -4658.766} C_VEL
LIN {X 0,Y 523.941,Z 285.216,A -85,B 0,C 180,E1 -4661.22,E2 -4661.22} C_VEL
LIN {X 0,Y 523.926,Z 285.222,A -85,B 0,C 180,E1 -4663.639,E2 -4663.639} C_VEL
LIN {X 0,Y 523.926,Z 285.225,A -85,B 0,C 180,E1 -4666.028,E2 -4666.028} C_VEL
LIN {X 0,Y 524.003,Z 285.211,A -85,B 0,C 180,E1 -4668.394,E2 -4668.394} C_VEL
LIN {X 0,Y 523.994,Z 285.21,A -85,B 0,C 180,E1 -4671.516,E2 -4671.516} C_VEL
LIN {X 0,Y 524.069,Z 285.202,A -85,B 0,C 180,E1 -4674.614,E2 -4674.614} C_VEL
LIN {X 0,Y 524.1,Z 285.197,A -85,B 0,C 180,E1 -4677.695,E2 -4677.695} C_VEL
LIN {X 0,Y 524.116,Z 285.196,A -85,B 0,C 180,E1 -4680.768,E2 -4680.768} C_VEL
LIN {X 0,Y 524.065,Z 285.2,A -85,B 0,C 180,E1 -4683.075,E2 -4683.075} C_VEL
LIN {X 0,Y 524.036,Z 285.208,A -85,B 0,C 180,E1 -4686.159,E2 -4686.159} C_VEL
LIN {X 0,Y 523.995,Z 285.209,A -85,B 0,C 180,E1 -4689.262,E2 -4689.262} C_VEL
LIN {X 0,Y 524,Z 285.207,A -85,B 0,C 180,E1 -4691.743,E2 -4691.743} C_VEL
LIN {X 0,Y 523.985,Z 285.214,A -85,B 0,C 180,E1 -4695.053,E2 -4695.053} C_VEL
LIN {X 0,Y 523.956,Z 285.213,A -85,B 0,C 180,E1 -4697.969,E2 -4697.969} C_VEL
LIN {X 0,Y 523.964,Z 285.215,A -85,B 0,C 180,E1 -4700.411,E2 -4700.411} C_VEL
LIN {X 0,Y 523.909,Z 285.228,A -85,B 0,C 180,E1 -4702.894,E2 -4702.894} C_VEL
LIN {X 0,Y 523.948,Z 285.217,A -85,B 0,C 180,E1 -4705.419,E2 -4705.419} C_VEL
LIN {X 0,Y 523.963,Z 285.212,A -85,B 0,C 180,E1 -4707.999,E2 -4707.999} C_VEL
LIN {X 0,Y 523.946,Z 285.219,A -85,B 0,C 180,E1 -4710.857,E2 -4710.857} C_VEL
LIN {X 0,Y 523.954,Z 285.215,A -85,B 0,C 180,E1 -4713.735,E2 -4713.735} C_VEL
LIN {X 0,Y 523.914,Z 285.218,A -85,B 0,C 180,E1 -4716.405,E2 -4716.405} C_VEL
LIN {X 0,Y 523.918,Z 285.223,A -85,B 0,C 180,E1 -4719.085,E2 -4719.085} C_VEL
LIN {X 0,Y 523.953,Z 285.214,A -85,B 0,C 180,E1 -4722.119,E2 -4722.119} C_VEL
LIN {X 0,Y 523.952,Z 285.22,A -85,B 0,C 180,E1 -4725.309,E2 -4725.309} C_VEL
LIN {X 0,Y 523.955,Z 285.213,A -85,B 0,C 180,E1 -4728.69,E2 -4728.69} C_VEL
LIN {X 0,Y 523.914,Z 285.22,A -85,B 0,C 180,E1 -4731.081,E2 -4731.081} C_VEL
LIN {X 0,Y 523.898,Z 285.229,A -85,B 0,C 180,E1 -4733.826,E2 -4733.826} C_VEL
LIN {X 0,Y 523.939,Z 285.215,A -85,B 0,C 180,E1 -4736.636,E2 -4736.636} C_VEL
LIN {X 0,Y 523.954,Z 285.215,A -85,B 0,C 180,E1 -4739.357,E2 -4739.357} C_VEL
LIN {X 0,Y 523.979,Z 285.217,A -85,B 0,C 180,E1 -4742.282,E2 -4742.282} C_VEL
LIN {X 0,Y 523.988,Z 285.28,A -85,B 0,C 180,E1 -4745.432,E2 -4745.432} C_VEL
LIN {X 0,Y 525.404,Z 293.248,A -85,B 0,C 180,E1 -4746.76,E2 -4746.76} C_VEL
LIN {X 0,Y 525.021,Z 311.645,A -85,B 0,C 180,E1 -4749.633,E2 -4749.633} C_VEL
LIN {X 0,Y 524.555,Z 331.319,A -85,B 0,C 180,E1 -4752.657,E2 -4752.657} C_VEL
LIN {X 0,Y 524.284,Z 345.707,A -85,B 0,C 180,E1 -4754.842,E2 -4754.842} C_VEL
LIN {X 0,Y 525.891,Z 356.669,A -85,B 0,C 180,E1 -4755.041,E2 -4755.041} C_VEL
LIN {X 0,Y 525.496,Z 453.988,A -85,B 0,C 180,E1 -4756.391,E2 -4756.391} C_VEL
LIN {X 0,Y 525.295,Z 467.296,A -85,B 0,C 180,E1 -4756.731,E2 -4756.731} C_VEL
LIN {X 0,Y 525.02,Z 479.484,A -85,B 0,C 180,E1 -4757.191,E2 -4757.191} C_VEL
LIN {X 0,Y 524.784,Z 491.533,A -85,B 0,C 180,E1 -4757.808,E2 -4757.808} C_VEL
LIN {X 0,Y 524.505,Z 503.405,A -85,B 0,C 180,E1 -4758.602,E2 -4758.602} C_VEL
LIN {X 0,Y 524.216,Z 513.867,A -85,B 0,C 180,E1 -4759.475,E2 -4759.475} C_VEL
LIN {X 0,Y 523.984,Z 522.422,A -85,B 0,C 180,E1 -4760.349,E2 -4760.349} C_VEL
LIN {X 0,Y 523.799,Z 530.318,A -85,B 0,C 180,E1 -4761.319,E2 -4761.319} C_VEL
LIN {X 0,Y 523.605,Z 538.029,A -85,B 0,C 180,E1 -4762.481,E2 -4762.481} C_VEL
LIN {X 0,Y 523.484,Z 545.138,A -85,B 0,C 180,E1 -4763.835,E2 -4763.835} C_VEL
LIN {X 0,Y 523.383,Z 549.867,A -85,B 0,C 180,E1 -4764.993,E2 -4764.993} C_VEL
LIN {X 0,Y 523.443,Z 553.484,A -85,B 0,C 180,E1 -4766.151,E2 -4766.151} C_VEL
LIN {X 0,Y 523.367,Z 555.346,A -85,B 0,C 180,E1 -4766.921,E2 -4766.921} C_VEL
LIN {X 0,Y 523.334,Z 556.743,A -85,B 0,C 180,E1 -4767.691,E2 -4767.691} C_VEL
LIN {X 0,Y 523.25,Z 558.345,A -85,B 0,C 180,E1 -4769.231,E2 -4769.231} C_VEL
LIN {X 0,Y 523.25,Z 558.561,A -85,B 0,C 180,E1 -4770,E2 -4770} C_VEL
LIN {X 0,Y 523.274,Z 557.737,A -85,B 0,C 180,E1 -4771.54,E2 -4771.54} C_VEL
LIN {X 0,Y 523.334,Z 556.741,A -85,B 0,C 180,E1 -4772.309,E2 -4772.309} C_VEL
LIN {X 0,Y 523.367,Z 555.343,A -85,B 0,C 180,E1 -4773.079,E2 -4773.079} C_VEL
LIN {X 0,Y 523.424,Z 552.403,A -85,B 0,C 180,E1 -4774.235,E2 -4774.235} C_VEL
LIN {X 0,Y 523.461,Z 548.422,A -85,B 0,C 180,E1 -4775.393,E2 -4775.393} C_VEL
